    |   movel([0.113074, -1.368242, -2.579336, -0.764810, 1.570796, 1.683871],accel_mss,speed_ms,0,blend_radius_m)
    |   movel([0.112842, -1.368148, -2.579401, -0.764840, 1.570796, 1.683639],accel_mss,speed_ms,0,blend_radius_m)
    |   movel([0.112523, -1.368181, -2.579379, -0.764830, 1.570796, 1.683319],accel_mss,speed_ms,0,blend_radius_m)
    |   movel([0.111949, -1.368213, -2.579357, -0.764820, 1.570796, 1.682746],accel_mss,speed_ms,0,blend_radius_m)
    |   movel([0.111243, -1.367988, -2.579512, -0.764890, 1.570796, 1.682039],accel_mss,speed_ms,0,blend_radius_m)
    |   movel([0.110603, -1.367616, -2.579767, -0.765006, 1.570796, 1.681399],accel_mss,speed_ms,0,blend_radius_m)
    |   movel([0.110212, -1.367165, -2.580077, -0.765147, 1.570796, 1.681008],accel_mss,speed_ms,0,blend_radius_m)
    |   movel([0.110029, -1.366891, -2.580265, -0.765233, 1.570796, 1.680825],accel_mss,speed_ms,0,blend_radius_m)
    |   movel([0.109878, -1.366752, -2.580361, -0.765276, 1.570796, 1.680674],accel_mss,speed_ms,0,blend_radius_m)
    |   movel([0.109999, -1.366376, -2.580619, -0.765394, 1.570796, 1.680795],accel_mss,speed_ms,0,blend_radius_m)
    |   movel([0.110066, -1.366058, -2.580837, -0.765494, 1.570796, 1.680862],accel_mss,speed_ms,0,blend_radius_m)
    |   movel([0.110125, -1.365664, -2.581106, -0.765618, 1.570796, 1.680922],accel_mss,speed_ms,0,blend_radius_m)
    |   movel([0.110214, -1.365078, -2.581508, -0.765803, 1.570796, 1.681011],accel_mss,speed_ms,0,blend_radius_m)
    |   movel([0.110312, -1.364717, -2.581755, -0.765918, 1.570796, 1.681108],accel_mss,speed_ms,0,blend_radius_m)
    |   movel([0.110471, -1.364372, -2.581990, -0.766027, 1.570796, 1.681267],accel_mss,speed_ms,0,blend_radius_m)
    |   movel([0.110770, -1.363875, -2.582330, -0.766185, 1.570796, 1.681566],accel_mss,speed_ms,0,blend_radius_m)
    |   movel([0.111001, -1.363529, -2.582566, -0.766294, 1.570796, 1.681797],accel_mss,speed_ms,0,blend_radius_m)
    |   movel([0.111258, -1.363172, -2.582809, -0.766408, 1.570796, 1.682054],accel_mss,speed_ms,0,blend_radius_m)
    |   movel([0.111508, -1.362853, -2.583026, -0.766510, 1.570796, 1.682304],accel_mss,speed_ms,0,blend_radius_m)
    |   movel([0.111700, -1.362635, -2.583174, -0.766579, 1.570796, 1.682497],accel_mss,speed_ms,0,blend_radius_m)
    |   movel([0.112170, -1.362219, -2.583458, -0.766713, 1.570796, 1.682966],accel_mss,speed_ms,0,blend_radius_m)
    |   movel([0.112837, -1.361736, -2.583786, -0.766867, 1.570796, 1.683634],accel_mss,speed_ms,0,blend_radius_m)
    |   movel([0.113532, -1.361295, -2.584086, -0.767009, 1.570796, 1.684329],accel_mss,speed_ms,0,blend_radius_m)
    |   movel([0.114080, -1.361022, -2.584271, -0.767097, 1.570796, 1.684876],accel_mss,speed_ms,0,blend_radius_m)
    |   movel([0.114439, -1.360855, -2.584384, -0.767150, 1.570796, 1.685235],accel_mss,speed_ms,0,blend_radius_m)
    |   movel([0.114838, -1.360572, -2.584576, -0.767242, 1.570796, 1.685635],accel_mss,speed_ms,0,blend_radius_m)
    |   movel([0.115414, -1.360389, -2.584700, -0.767301, 1.570796, 1.686211],accel_mss,speed_ms,0,blend_radius_m)
    |   movel([0.115941, -1.360262, -2.584785, -0.767341, 1.570796, 1.686737],accel_mss,speed_ms,0,blend_radius_m)
    |   movel([0.116093, -1.360400, -2.584692, -0.767297, 1.570796, 1.686889],accel_mss,speed_ms,0,blend_radius_m)
    |   movel([0.116466, -1.360370, -2.584712, -0.767307, 1.570796, 1.687262],accel_mss,speed_ms,0,blend_radius_m)
    |   movel([0.117091, -1.360338, -2.584734, -0.767317, 1.570796, 1.687887],accel_mss,speed_ms,0,blend_radius_m)
    |   movel([0.117773, -1.360429, -2.584672, -0.767288, 1.570796, 1.688569],accel_mss,speed_ms,0,blend_radius_m)
    |   movel([0.118423, -1.360624, -2.584540, -0.767225, 1.570796, 1.689219],accel_mss,speed_ms,0,blend_radius_m)
    |   movel([0.118955, -1.360908, -2.584348, -0.767133, 1.570796, 1.689751],accel_mss,speed_ms,0,blend_radius_m)
    |   movel([0.119345, -1.361234, -2.584126, -0.767028, 1.570796, 1.690142],accel_mss,speed_ms,0,blend_radius_m)
    |   movel([0.119677, -1.361646, -2.583847, -0.766896, 1.570796, 1.690474],accel_mss,speed_ms,0,blend_radius_m)
    |   movel([0.119903, -1.362061, -2.583565, -0.766763, 1.570796, 1.690699],accel_mss,speed_ms,0,blend_radius_m)
    |   movel([0.119940, -1.362378, -2.583349, -0.766661, 1.570796, 1.690737],accel_mss,speed_ms,0,blend_radius_m)
    |   movel([0.119963, -1.362607, -2.583194, -0.766588, 1.570796, 1.690759],accel_mss,speed_ms,0,blend_radius_m)
    |   movel([0.120018, -1.362814, -2.583053, -0.766522, 1.570796, 1.690814],accel_mss,speed_ms,0,blend_radius_m)
    |   movel([0.119974, -1.363148, -2.582825, -0.766416, 1.570796, 1.690771],accel_mss,speed_ms,0,blend_radius_m)
    |   movel([0.119941, -1.363465, -2.582609, -0.766315, 1.570796, 1.690737],accel_mss,speed_ms,0,blend_radius_m)
    |   movel([0.120103, -1.363586, -2.582526, -0.766276, 1.570796, 1.690899],accel_mss,speed_ms,0,blend_radius_m)
    |   movel([0.120063, -1.363825, -2.582364, -0.766200, 1.570796, 1.690859],accel_mss,speed_ms,0,blend_radius_m)
    |   movel([0.119744, -1.364111, -2.582168, -0.766109, 1.570796, 1.690540],accel_mss,speed_ms,0,blend_radius_m)
    |   movel([0.119488, -1.364550, -2.581869, -0.765970, 1.570796, 1.690284],accel_mss,speed_ms,0,blend_radius_m)
    |   movel([0.118959, -1.365356, -2.581317, -0.765715, 1.570796, 1.689756],accel_mss,speed_ms,0,blend_radius_m)
    |   movel([0.118185, -1.366126, -2.580790, -0.765473, 1.570796, 1.688981],accel_mss,speed_ms,0,blend_radius_m)
    |   movel([0.117294, -1.366745, -2.580366, -0.765279, 1.570796, 1.688091],accel_mss,speed_ms,0,blend_radius_m)
    |   movel([0.116416, -1.367114, -2.580112, -0.765163, 1.570796, 1.687213],accel_mss,speed_ms,0,blend_radius_m)
    |   movel([0.116092, -1.367241, -2.580025, -0.765123, 1.570796, 1.686888],accel_mss,speed_ms,0,blend_radius_m)
    |   movel([0.115731, -1.367579, -2.579793, -0.765017, 1.570796, 1.686528],accel_mss,speed_ms,0,blend_radius_m)
    |   movel([0.115661, -1.367816, -2.579630, -0.764943, 1.570796, 1.686457],accel_mss,speed_ms,0,blend_radius_m)
    |   movel([0.115748, -1.368044, -2.579473, -0.764872, 1.570796, 1.686544],accel_mss,speed_ms,0,blend_radius_m)
    |   movel([0.115829, -1.368244, -2.579335, -0.764810, 1.570796, 1.686625],accel_mss,speed_ms,0,blend_radius_m)
    |   movel([0.115565, -1.368425, -2.579211, -0.764754, 1.570796, 1.686362],accel_mss,speed_ms,0,blend_radius_m)
    |   movel([0.115373, -1.368755, -2.578983, -0.764651, 1.570796, 1.686169],accel_mss,speed_ms,0,blend_radius_m)
    |   movel([0.115111, -1.368926, -2.578865, -0.764598, 1.570796, 1.685907],accel_mss,speed_ms,0,blend_radius_m)
    |   movel([0.114895, -1.368883, -2.578895, -0.764611, 1.570796, 1.685691],accel_mss,speed_ms,0,blend_radius_m)
    |   movel([0.114646, -1.368902, -2.578882, -0.764605, 1.570796, 1.685442],accel_mss,speed_ms,0,blend_radius_m)
    |   movel([0.114354, -1.368984, -2.578826, -0.764580, 1.570796, 1.685151],accel_mss,speed_ms,0,blend_radius_m)
    |   movel([0.114218, -1.368703, -2.579019, -0.764667, 1.570796, 1.685014],accel_mss,speed_ms,0,blend_radius_m)
    |   movel([0.114179, -1.368458, -2.579188, -0.764743, 1.570796, 1.684976],accel_mss,speed_ms,0,blend_radius_m)
    |   movel([0.113902, -1.368506, -2.579155, -0.764728, 1.570796, 1.684698],accel_mss,speed_ms,0,blend_radius_m)
    |   movel([0.113822, -1.368763, -2.578978, -0.764649, 1.570796, 1.684618],accel_mss,speed_ms,0,blend_radius_m)
    |   movel([0.113746, -1.369031, -2.578793, -0.764565, 1.570796, 1.684542],accel_mss,speed_ms,0,blend_radius_m)
    |   movel([0.113433, -1.369351, -2.578572, -0.764466, 1.570796, 1.684229],accel_mss,speed_ms,0,blend_radius_m)
    |   speed_ms = 0.003
    |   movel([0.113433, -1.372674, -2.580076, -0.759639, 1.570796, 1.684229],accel_mss,speed_ms,0,blend_radius_m)
    |   speed_ms = 0.007
    |   movel([0.113200, -1.372440, -2.580238, -0.759711, 1.570796, 1.683996],accel_mss,speed_ms,0,blend_radius_m)
    |   movel([0.113209, -1.372110, -2.580467, -0.759812, 1.570796, 1.684005],accel_mss,speed_ms,0,blend_radius_m)
    |   movel([0.113200, -1.371785, -2.580692, -0.759912, 1.570796, 1.683996],accel_mss,speed_ms,0,blend_radius_m)
    |   movel([0.113074, -1.371568, -2.580842, -0.759979, 1.570796, 1.683871],accel_mss,speed_ms,0,blend_radius_m)
    |   movel([0.112842, -1.371474, -2.580907, -0.760008, 1.570796, 1.683639],accel_mss,speed_ms,0,blend_radius_m)
    |   movel([0.112523, -1.371507, -2.580885, -0.759998, 1.570796, 1.683319],accel_mss,speed_ms,0,blend_radius_m)
    |   movel([0.111949, -1.371539, -2.580863, -0.759988, 1.570796, 1.682746],accel_mss,speed_ms,0,blend_radius_m)
    |   movel([0.111243, -1.371314, -2.581018, -0.760057, 1.570796, 1.682039],accel_mss,speed_ms,0,blend_radius_m)
    |   movel([0.110603, -1.370943, -2.581274, -0.760171, 1.570796, 1.681399],accel_mss,speed_ms,0,blend_radius_m)
    |   movel([0.110212, -1.370493, -2.581585, -0.760311, 1.570796, 1.681008],accel_mss,speed_ms,0,blend_radius_m)
    |   movel([0.110029, -1.370220, -2.581773, -0.760395, 1.570796, 1.680825],accel_mss,speed_ms,0,blend_radius_m)
    |   movel([0.109878, -1.370081, -2.581869, -0.760438, 1.570796, 1.680674],accel_mss,speed_ms,0,blend_radius_m)
    |   movel([0.109999, -1.369706, -2.582128, -0.760555, 1.570796, 1.680795],accel_mss,speed_ms,0,blend_radius_m)
    |   movel([0.110066, -1.369389, -2.582347, -0.760653, 1.570796, 1.680862],accel_mss,speed_ms,0,blend_radius_m)
    |   movel([0.110125, -1.368997, -2.582617, -0.760776, 1.570796, 1.680922],accel_mss,speed_ms,0,blend_radius_m)
    |   movel([0.110214, -1.368412, -2.583019, -0.760958, 1.570796, 1.681011],accel_mss,speed_ms,0,blend_radius_m)
    |   movel([0.110312, -1.368052, -2.583266, -0.761071, 1.570796, 1.681108],accel_mss,speed_ms,0,blend_radius_m)
    |   movel([0.110471, -1.367708, -2.583502, -0.761178, 1.570796, 1.681267],accel_mss,speed_ms,0,blend_radius_m)
    |   movel([0.110770, -1.367212, -2.583843, -0.761334, 1.570796, 1.681566],accel_mss,speed_ms,0,blend_radius_m)
    |   movel([0.111001, -1.366867, -2.584079, -0.761443, 1.570796, 1.681797],accel_mss,speed_ms,0,blend_radius_m)
    |   movel([0.111258, -1.366511, -2.584323, -0.761555, 1.570796, 1.682054],accel_mss,speed_ms,0,blend_radius_m)
    |   movel([0.111508, -1.366193, -2.584541, -0.761655, 1.570796, 1.682304],accel_mss,speed_ms,0,blend_radius_m)
    |   movel([0.111700, -1.365976, -2.584689, -0.761724, 1.570796, 1.682497],accel_mss,speed_ms,0,blend_radius_m)
    |   movel([0.112170, -1.365560, -2.584974, -0.761855, 1.570796, 1.682966],accel_mss,speed_ms,0,blend_radius_m)
    |   movel([0.112837, -1.365078, -2.585303, -0.762008, 1.570796, 1.683634],accel_mss,speed_ms,0,blend_radius_m)
    |   movel([0.113532, -1.364639, -2.585603, -0.762147, 1.570796, 1.684329],accel_mss,speed_ms,0,blend_radius_m)
    |   movel([0.114080, -1.364366, -2.585789, -0.762234, 1.570796, 1.684876],accel_mss,speed_ms,0,blend_radius_m)
    |   movel([0.114439, -1.364200, -2.585902, -0.762287, 1.570796, 1.685235],accel_mss,speed_ms,0,blend_radius_m)
    |   movel([0.114838, -1.363918, -2.586094, -0.762377, 1.570796, 1.685635],accel_mss,speed_ms,0,blend_radius_m)
    |   movel([0.115414, -1.363735, -2.586219, -0.762435, 1.570796, 1.686211],accel_mss,speed_ms,0,blend_radius_m)
    |   movel([0.115941, -1.363609, -2.586304, -0.762475, 1.570796, 1.686737],accel_mss,speed_ms,0,blend_radius_m)
    |   movel([0.116093, -1.363746, -2.586211, -0.762432, 1.570796, 1.686889],accel_mss,speed_ms,0,blend_radius_m)
    |   movel([0.116466, -1.363716, -2.586231, -0.762441, 1.570796, 1.687262],accel_mss,speed_ms,0,blend_radius_m)
    |   movel([0.117091, -1.363685, -2.586253, -0.762451, 1.570796, 1.687887],accel_mss,speed_ms,0,blend_radius_m)
    |   movel([0.117773, -1.363775, -2.586191, -0.762422, 1.570796, 1.688569],accel_mss,speed_ms,0,blend_radius_m)
    |   movel([0.118423, -1.363970, -2.586059, -0.762360, 1.570796, 1.689219],accel_mss,speed_ms,0,blend_radius_m)
    |   movel([0.118955, -1.364253, -2.585866, -0.762270, 1.570796, 1.689751],accel_mss,speed_ms,0,blend_radius_m)
    |   movel([0.119345, -1.364579, -2.585644, -0.762167, 1.570796, 1.690142],accel_mss,speed_ms,0,blend_radius_m)
    |   movel([0.119677, -1.364989, -2.585364, -0.762036, 1.570796, 1.690474],accel_mss,speed_ms,0,blend_radius_m)
    |   movel([0.119903, -1.365403, -2.585081, -0.761905, 1.570796, 1.690699],accel_mss,speed_ms,0,blend_radius_m)
    |   movel([0.119940, -1.365720, -2.584865, -0.761805, 1.570796, 1.690737],accel_mss,speed_ms,0,blend_radius_m)
    |   movel([0.119963, -1.365947, -2.584709, -0.761733, 1.570796, 1.690759],accel_mss,speed_ms,0,blend_radius_m)
    |   movel([0.120018, -1.366154, -2.584568, -0.761667, 1.570796, 1.690814],accel_mss,speed_ms,0,blend_radius_m)
    |   movel([0.119974, -1.366487, -2.584339, -0.761562, 1.570796, 1.690771],accel_mss,speed_ms,0,blend_radius_m)
    |   movel([0.119941, -1.366803, -2.584123, -0.761463, 1.570796, 1.690737],accel_mss,speed_ms,0,blend_radius_m)
    |   movel([0.120103, -1.366924, -2.584040, -0.761425, 1.570796, 1.690899],accel_mss,speed_ms,0,blend_radius_m)
    |   movel([0.120063, -1.367162, -2.583877, -0.761350, 1.570796, 1.690859],accel_mss,speed_ms,0,blend_radius_m)
    |   movel([0.119744, -1.367448, -2.583681, -0.761260, 1.570796, 1.690540],accel_mss,speed_ms,0,blend_radius_m)
    |   movel([0.119488, -1.367886, -2.583381, -0.761123, 1.570796, 1.690284],accel_mss,speed_ms,0,blend_radius_m)
    |   movel([0.118959, -1.368690, -2.582828, -0.760871, 1.570796, 1.689756],accel_mss,speed_ms,0,blend_radius_m)
    |   movel([0.118185, -1.369457, -2.582300, -0.760632, 1.570796, 1.688981],accel_mss,speed_ms,0,blend_radius_m)
    |   movel([0.117294, -1.370074, -2.581874, -0.760441, 1.570796, 1.688091],accel_mss,speed_ms,0,blend_radius_m)
    |   movel([0.116416, -1.370443, -2.581620, -0.760326, 1.570796, 1.687213],accel_mss,speed_ms,0,blend_radius_m)
    |   movel([0.116092, -1.370570, -2.581532, -0.760287, 1.570796, 1.686888],accel_mss,speed_ms,0,blend_radius_m)
    |   movel([0.115731, -1.370906, -2.581300, -0.760183, 1.570796, 1.686528],accel_mss,speed_ms,0,blend_radius_m)
    |   movel([0.115661, -1.371143, -2.581136, -0.760110, 1.570796, 1.686457],accel_mss,speed_ms,0,blend_radius_m)
    |   movel([0.115748, -1.371370, -2.580979, -0.760040, 1.570796, 1.686544],accel_mss,speed_ms,0,blend_radius_m)
    |   movel([0.115829, -1.371570, -2.580841, -0.759978, 1.570796, 1.686625],accel_mss,speed_ms,0,blend_radius_m)
    |   movel([0.115565, -1.371750, -2.580716, -0.759923, 1.570796, 1.686362],accel_mss,speed_ms,0,blend_radius_m)
    |   movel([0.115373, -1.372079, -2.580488, -0.759822, 1.570796, 1.686169],accel_mss,speed_ms,0,blend_radius_m)
    |   movel([0.115111, -1.372250, -2.580370, -0.759769, 1.570796, 1.685907],accel_mss,speed_ms,0,blend_radius_m)
    |   movel([0.114895, -1.372207, -2.580400, -0.759782, 1.570796, 1.685691],accel_mss,speed_ms,0,blend_radius_m)
    |   movel([0.114646, -1.372226, -2.580387, -0.759777, 1.570796, 1.685442],accel_mss,speed_ms,0,blend_radius_m)
    |   movel([0.114354, -1.372307, -2.580330, -0.759751, 1.570796, 1.685151],accel_mss,speed_ms,0,blend_radius_m)
    |   movel([0.114218, -1.372028, -2.580524, -0.759837, 1.570796, 1.685014],accel_mss,speed_ms,0,blend_radius_m)
    |   movel([0.114179, -1.371783, -2.580693, -0.759913, 1.570796, 1.684976],accel_mss,speed_ms,0,blend_radius_m)
    |   movel([0.113902, -1.371831, -2.580660, -0.759898, 1.570796, 1.684698],accel_mss,speed_ms,0,blend_radius_m)
    |   movel([0.113822, -1.372087, -2.580483, -0.759819, 1.570796, 1.684618],accel_mss,speed_ms,0,blend_radius_m)
    |   movel([0.113746, -1.372354, -2.580298, -0.759737, 1.570796, 1.684542],accel_mss,speed_ms,0,blend_radius_m)
    |   movel([0.113433, -1.372674, -2.580076, -0.759639, 1.570796, 1.684229],accel_mss,speed_ms,0,blend_radius_m)
    |   speed_ms = 0.003
    |   movel([0.113433, -1.359522, -2.574009, -0.778858, 1.570796, 1.684229],accel_mss,speed_ms,0,blend_radius_m)
    |   speed_ms = 1.000
    |   movel([0.113433, -1.334323, -2.561482, -0.816584, 1.570796, 1.684229],accel_mss,speed_ms,0,blend_radius_m)
    |   movel([0.114853, -1.333089, -2.562290, -0.817010, 1.570796, 1.685649],accel_mss,speed_ms,0,blend_radius_m)
    |   movel([0.114853, -1.358310, -2.574833, -0.779247, 1.570796, 1.685649],accel_mss,speed_ms,0,blend_radius_m)
    |   speed_ms = 0.003
    |   movel([0.114853, -1.368148, -2.579401, -0.764840, 1.570796, 1.685649],accel_mss,speed_ms,0,blend_radius_m)
    |   speed_ms = 0.007
    |   movel([0.114797, -1.367902, -2.579570, -0.764916, 1.570796, 1.685593],accel_mss,speed_ms,0,blend_radius_m)
    |   movel([0.114829, -1.367601, -2.579777, -0.765011, 1.570796, 1.685626],accel_mss,speed_ms,0,blend_radius_m)
    |   movel([0.114890, -1.367234, -2.580030, -0.765125, 1.570796, 1.685686],accel_mss,speed_ms,0,blend_radius_m)
    |   movel([0.115073, -1.366962, -2.580217, -0.765211, 1.570796, 1.685869],accel_mss,speed_ms,0,blend_radius_m)
    |   movel([0.115228, -1.367178, -2.580068, -0.765143, 1.570796, 1.686024],accel_mss,speed_ms,0,blend_radius_m)
    |   movel([0.115200, -1.367570, -2.579799, -0.765020, 1.570796, 1.685996],accel_mss,speed_ms,0,blend_radius_m)
    |   movel([0.115155, -1.367837, -2.579615, -0.764937, 1.570796, 1.685951],accel_mss,speed_ms,0,blend_radius_m)
    |   movel([0.115032, -1.368103, -2.579432, -0.764854, 1.570796, 1.685828],accel_mss,speed_ms,0,blend_radius_m)
    |   speed_ms = 0.003
    |   movel([0.114853, -1.371474, -2.580907, -0.760008, 1.570796, 1.685649],accel_mss,speed_ms,0,blend_radius_m)
    |   speed_ms = 0.007
    |   movel([0.114797, -1.371229, -2.581077, -0.760083, 1.570796, 1.685593],accel_mss,speed_ms,0,blend_radius_m)
    |   movel([0.114829, -1.370928, -2.581285, -0.760176, 1.570796, 1.685626],accel_mss,speed_ms,0,blend_radius_m)
    |   movel([0.114890, -1.370562, -2.581537, -0.760289, 1.570796, 1.685686],accel_mss,speed_ms,0,blend_radius_m)
    |   movel([0.115073, -1.370291, -2.581725, -0.760373, 1.570796, 1.685869],accel_mss,speed_ms,0,blend_radius_m)
    |   movel([0.115228, -1.370506, -2.581576, -0.760307, 1.570796, 1.686024],accel_mss,speed_ms,0,blend_radius_m)
    |   movel([0.115200, -1.370898, -2.581306, -0.760186, 1.570796, 1.685996],accel_mss,speed_ms,0,blend_radius_m)
    |   movel([0.115155, -1.371163, -2.581122, -0.760104, 1.570796, 1.685951],accel_mss,speed_ms,0,blend_radius_m)
    |   movel([0.115032, -1.371429, -2.580938, -0.760022, 1.570796, 1.685828],accel_mss,speed_ms,0,blend_radius_m)
    |   speed_ms = 0.003
    |   movel([0.114853, -1.358310, -2.574833, -0.779247, 1.570796, 1.685649],accel_mss,speed_ms,0,blend_radius_m)
    |   speed_ms = 1.000
    |   movel([0.114853, -1.333089, -2.562290, -0.817010, 1.570796, 1.685649],accel_mss,speed_ms,0,blend_radius_m)
    |   movel([0.115300, -1.331245, -2.563492, -0.817651, 1.570796, 1.686097],accel_mss,speed_ms,0,blend_radius_m)
    |   movel([0.115300, -1.356498, -2.576059, -0.779832, 1.570796, 1.686097],accel_mss,speed_ms,0,blend_radius_m)
    |   speed_ms = 0.003
    |   movel([0.115300, -1.366350, -2.580637, -0.765403, 1.570796, 1.686097],accel_mss,speed_ms,0,blend_radius_m)
    |   speed_ms = 0.007
    |   movel([0.115147, -1.366199, -2.580740, -0.765450, 1.570796, 1.685943],accel_mss,speed_ms,0,blend_radius_m)
    |   movel([0.115161, -1.365756, -2.581044, -0.765589, 1.570796, 1.685958],accel_mss,speed_ms,0,blend_radius_m)
    |   movel([0.114937, -1.365561, -2.581178, -0.765651, 1.570796, 1.685734],accel_mss,speed_ms,0,blend_radius_m)
    |   movel([0.114685, -1.365743, -2.581052, -0.765593, 1.570796, 1.685482],accel_mss,speed_ms,0,blend_radius_m)
    |   movel([0.114564, -1.365999, -2.580877, -0.765513, 1.570796, 1.685360],accel_mss,speed_ms,0,blend_radius_m)
    |   movel([0.114505, -1.366260, -2.580699, -0.765431, 1.570796, 1.685301],accel_mss,speed_ms,0,blend_radius_m)
    |   movel([0.114305, -1.366479, -2.580548, -0.765362, 1.570796, 1.685101],accel_mss,speed_ms,0,blend_radius_m)
    |   movel([0.114150, -1.366331, -2.580649, -0.765408, 1.570796, 1.684947],accel_mss,speed_ms,0,blend_radius_m)
    |   movel([0.114152, -1.365911, -2.580937, -0.765540, 1.570796, 1.684948],accel_mss,speed_ms,0,blend_radius_m)
    |   movel([0.114050, -1.365717, -2.581071, -0.765602, 1.570796, 1.684846],accel_mss,speed_ms,0,blend_radius_m)
    |   movel([0.113872, -1.365616, -2.581140, -0.765634, 1.570796, 1.684668],accel_mss,speed_ms,0,blend_radius_m)
    |   movel([0.113440, -1.365643, -2.581121, -0.765625, 1.570796, 1.684236],accel_mss,speed_ms,0,blend_radius_m)
    |   movel([0.113058, -1.365470, -2.581240, -0.765680, 1.570796, 1.683854],accel_mss,speed_ms,0,blend_radius_m)
    |   movel([0.112877, -1.365278, -2.581371, -0.765740, 1.570796, 1.683673],accel_mss,speed_ms,0,blend_radius_m)
    |   movel([0.112754, -1.365018, -2.581549, -0.765822, 1.570796, 1.683550],accel_mss,speed_ms,0,blend_radius_m)
    |   movel([0.112941, -1.364690, -2.581773, -0.765926, 1.570796, 1.683737],accel_mss,speed_ms,0,blend_radius_m)
    |   movel([0.113216, -1.364401, -2.581970, -0.766017, 1.570796, 1.684013],accel_mss,speed_ms,0,blend_radius_m)
    |   movel([0.113587, -1.364309, -2.582033, -0.766047, 1.570796, 1.684383],accel_mss,speed_ms,0,blend_radius_m)
    |   movel([0.113919, -1.364304, -2.582037, -0.766048, 1.570796, 1.684715],accel_mss,speed_ms,0,blend_radius_m)
    |   movel([0.114137, -1.364361, -2.581997, -0.766030, 1.570796, 1.684933],accel_mss,speed_ms,0,blend_radius_m)
    |   movel([0.114307, -1.364503, -2.581901, -0.765985, 1.570796, 1.685103],accel_mss,speed_ms,0,blend_radius_m)
    |   movel([0.114482, -1.364779, -2.581712, -0.765898, 1.570796, 1.685278],accel_mss,speed_ms,0,blend_radius_m)
    |   movel([0.114658, -1.365037, -2.581536, -0.765816, 1.570796, 1.685455],accel_mss,speed_ms,0,blend_radius_m)
    |   movel([0.114837, -1.365132, -2.581471, -0.765786, 1.570796, 1.685633],accel_mss,speed_ms,0,blend_radius_m)
    |   movel([0.115325, -1.364910, -2.581623, -0.765856, 1.570796, 1.686121],accel_mss,speed_ms,0,blend_radius_m)
    |   movel([0.115621, -1.364725, -2.581749, -0.765915, 1.570796, 1.686417],accel_mss,speed_ms,0,blend_radius_m)
    |   movel([0.115907, -1.364643, -2.581805, -0.765941, 1.570796, 1.686703],accel_mss,speed_ms,0,blend_radius_m)
    |   movel([0.116371, -1.364357, -2.582001, -0.766032, 1.570796, 1.687167],accel_mss,speed_ms,0,blend_radius_m)
    |   movel([0.116464, -1.364121, -2.582162, -0.766106, 1.570796, 1.687260],accel_mss,speed_ms,0,blend_radius_m)
    |   movel([0.116312, -1.363881, -2.582325, -0.766182, 1.570796, 1.687108],accel_mss,speed_ms,0,blend_radius_m)
    |   movel([0.116012, -1.364107, -2.582171, -0.766111, 1.570796, 1.686808],accel_mss,speed_ms,0,blend_radius_m)
    |   movel([0.115646, -1.364425, -2.581954, -0.766010, 1.570796, 1.686443],accel_mss,speed_ms,0,blend_radius_m)
    |   movel([0.115581, -1.364176, -2.582124, -0.766089, 1.570796, 1.686377],accel_mss,speed_ms,0,blend_radius_m)
    |   movel([0.115831, -1.363884, -2.582323, -0.766181, 1.570796, 1.686627],accel_mss,speed_ms,0,blend_radius_m)
    |   movel([0.116106, -1.363605, -2.582514, -0.766270, 1.570796, 1.686902],accel_mss,speed_ms,0,blend_radius_m)
    |   movel([0.116442, -1.363532, -2.582564, -0.766294, 1.570796, 1.687238],accel_mss,speed_ms,0,blend_radius_m)
    |   movel([0.116664, -1.363637, -2.582492, -0.766260, 1.570796, 1.687460],accel_mss,speed_ms,0,blend_radius_m)
    |   movel([0.116856, -1.363863, -2.582338, -0.766188, 1.570796, 1.687653],accel_mss,speed_ms,0,blend_radius_m)
    |   movel([0.116823, -1.364149, -2.582142, -0.766097, 1.570796, 1.687619],accel_mss,speed_ms,0,blend_radius_m)
    |   movel([0.116538, -1.364541, -2.581875, -0.765973, 1.570796, 1.687334],accel_mss,speed_ms,0,blend_radius_m)
    |   movel([0.115912, -1.365137, -2.581468, -0.765785, 1.570796, 1.686708],accel_mss,speed_ms,0,blend_radius_m)
    |   movel([0.115665, -1.365447, -2.581255, -0.765687, 1.570796, 1.686461],accel_mss,speed_ms,0,blend_radius_m)
    |   movel([0.115550, -1.365853, -2.580977, -0.765559, 1.570796, 1.686346],accel_mss,speed_ms,0,blend_radius_m)
    |   movel([0.115461, -1.366207, -2.580735, -0.765447, 1.570796, 1.686258],accel_mss,speed_ms,0,blend_radius_m)
    |   speed_ms = 0.003
    |   movel([0.115300, -1.369680, -2.582146, -0.760563, 1.570796, 1.686097],accel_mss,speed_ms,0,blend_radius_m)
    |   speed_ms = 0.007
    |   movel([0.115147, -1.369530, -2.582249, -0.760610, 1.570796, 1.685943],accel_mss,speed_ms,0,blend_radius_m)
    |   movel([0.115161, -1.369088, -2.582554, -0.760747, 1.570796, 1.685958],accel_mss,speed_ms,0,blend_radius_m)
    |   movel([0.114937, -1.368893, -2.582688, -0.760808, 1.570796, 1.685734],accel_mss,speed_ms,0,blend_radius_m)
    |   movel([0.114685, -1.369075, -2.582562, -0.760751, 1.570796, 1.685482],accel_mss,speed_ms,0,blend_radius_m)
    |   movel([0.114564, -1.369331, -2.582387, -0.760671, 1.570796, 1.685360],accel_mss,speed_ms,0,blend_radius_m)
    |   movel([0.114505, -1.369590, -2.582208, -0.760591, 1.570796, 1.685301],accel_mss,speed_ms,0,blend_radius_m)
    |   movel([0.114305, -1.369810, -2.582057, -0.760523, 1.570796, 1.685101],accel_mss,speed_ms,0,blend_radius_m)
    |   movel([0.114150, -1.369662, -2.582158, -0.760569, 1.570796, 1.684947],accel_mss,speed_ms,0,blend_radius_m)
    |   movel([0.114152, -1.369243, -2.582447, -0.760699, 1.570796, 1.684948],accel_mss,speed_ms,0,blend_radius_m)
    |   movel([0.114050, -1.369049, -2.582581, -0.760759, 1.570796, 1.684846],accel_mss,speed_ms,0,blend_radius_m)
    |   movel([0.113872, -1.368948, -2.582650, -0.760791, 1.570796, 1.684668],accel_mss,speed_ms,0,blend_radius_m)
    |   movel([0.113440, -1.368975, -2.582631, -0.760782, 1.570796, 1.684236],accel_mss,speed_ms,0,blend_radius_m)
    |   movel([0.113058, -1.368803, -2.582750, -0.760836, 1.570796, 1.683854],accel_mss,speed_ms,0,blend_radius_m)
    |   movel([0.112877, -1.368611, -2.582882, -0.760896, 1.570796, 1.683673],accel_mss,speed_ms,0,blend_radius_m)
    |   movel([0.112754, -1.368352, -2.583060, -0.760977, 1.570796, 1.683550],accel_mss,speed_ms,0,blend_radius_m)
    |   movel([0.112941, -1.368025, -2.583285, -0.761079, 1.570796, 1.683737],accel_mss,speed_ms,0,blend_radius_m)
    |   movel([0.113216, -1.367737, -2.583483, -0.761169, 1.570796, 1.684013],accel_mss,speed_ms,0,blend_radius_m)
    |   movel([0.113587, -1.367646, -2.583545, -0.761198, 1.570796, 1.684383],accel_mss,speed_ms,0,blend_radius_m)
    |   movel([0.113919, -1.367640, -2.583549, -0.761200, 1.570796, 1.684715],accel_mss,speed_ms,0,blend_radius_m)
    |   movel([0.114137, -1.367697, -2.583510, -0.761182, 1.570796, 1.684933],accel_mss,speed_ms,0,blend_radius_m)
    |   movel([0.114307, -1.367839, -2.583413, -0.761137, 1.570796, 1.685103],accel_mss,speed_ms,0,blend_radius_m)
    |   movel([0.114482, -1.368114, -2.583224, -0.761051, 1.570796, 1.685278],accel_mss,speed_ms,0,blend_radius_m)
    |   movel([0.114658, -1.368371, -2.583047, -0.760971, 1.570796, 1.685455],accel_mss,speed_ms,0,blend_radius_m)
    |   movel([0.114837, -1.368465, -2.582982, -0.760941, 1.570796, 1.685633],accel_mss,speed_ms,0,blend_radius_m)
    |   movel([0.115325, -1.368244, -2.583134, -0.761011, 1.570796, 1.686121],accel_mss,speed_ms,0,blend_radius_m)
    |   movel([0.115621, -1.368060, -2.583261, -0.761068, 1.570796, 1.686417],accel_mss,speed_ms,0,blend_radius_m)
    |   movel([0.115907, -1.367978, -2.583317, -0.761094, 1.570796, 1.686703],accel_mss,speed_ms,0,blend_radius_m)
    |   movel([0.116371, -1.367693, -2.583513, -0.761183, 1.570796, 1.687167],accel_mss,speed_ms,0,blend_radius_m)
    |   movel([0.116464, -1.367457, -2.583675, -0.761257, 1.570796, 1.687260],accel_mss,speed_ms,0,blend_radius_m)
    |   movel([0.116312, -1.367218, -2.583838, -0.761332, 1.570796, 1.687108],accel_mss,speed_ms,0,blend_radius_m)
    |   movel([0.116012, -1.367444, -2.583684, -0.761261, 1.570796, 1.686808],accel_mss,speed_ms,0,blend_radius_m)
    |   movel([0.115646, -1.367760, -2.583467, -0.761162, 1.570796, 1.686443],accel_mss,speed_ms,0,blend_radius_m)
    |   movel([0.115581, -1.367513, -2.583637, -0.761240, 1.570796, 1.686377],accel_mss,speed_ms,0,blend_radius_m)
    |   movel([0.115831, -1.367222, -2.583836, -0.761331, 1.570796, 1.686627],accel_mss,speed_ms,0,blend_radius_m)
    |   movel([0.116106, -1.366943, -2.584028, -0.761419, 1.570796, 1.686902],accel_mss,speed_ms,0,blend_radius_m)
    |   movel([0.116442, -1.366870, -2.584077, -0.761442, 1.570796, 1.687238],accel_mss,speed_ms,0,blend_radius_m)
    |   movel([0.116664, -1.366974, -2.584006, -0.761409, 1.570796, 1.687460],accel_mss,speed_ms,0,blend_radius_m)
    |   movel([0.116856, -1.367200, -2.583851, -0.761338, 1.570796, 1.687653],accel_mss,speed_ms,0,blend_radius_m)
    |   movel([0.116823, -1.367486, -2.583655, -0.761248, 1.570796, 1.687619],accel_mss,speed_ms,0,blend_radius_m)
    |   movel([0.116538, -1.367876, -2.583387, -0.761126, 1.570796, 1.687334],accel_mss,speed_ms,0,blend_radius_m)
    |   movel([0.115912, -1.368471, -2.582979, -0.760940, 1.570796, 1.686708],accel_mss,speed_ms,0,blend_radius_m)
    |   movel([0.115665, -1.368780, -2.582766, -0.760843, 1.570796, 1.686461],accel_mss,speed_ms,0,blend_radius_m)
    |   movel([0.115550, -1.369185, -2.582487, -0.760717, 1.570796, 1.686346],accel_mss,speed_ms,0,blend_radius_m)
    |   movel([0.115461, -1.369538, -2.582244, -0.760607, 1.570796, 1.686258],accel_mss,speed_ms,0,blend_radius_m)
    |   speed_ms = 0.003
    |   movel([0.115300, -1.356498, -2.576059, -0.779832, 1.570796, 1.686097],accel_mss,speed_ms,0,blend_radius_m)
    |   speed_ms = 1.000
    |   movel([0.115300, -1.331245, -2.563492, -0.817651, 1.570796, 1.686097],accel_mss,speed_ms,0,blend_radius_m)
    |   movel([0.114036, -1.330032, -2.564282, -0.818075, 1.570796, 1.684833],accel_mss,speed_ms,0,blend_radius_m)
    |   movel([0.114036, -1.355305, -2.576864, -0.780220, 1.570796, 1.684833],accel_mss,speed_ms,0,blend_radius_m)
    |   speed_ms = 0.003
    |   movel([0.114036, -1.365165, -2.581448, -0.765776, 1.570796, 1.684833],accel_mss,speed_ms,0,blend_radius_m)
    |   speed_ms = 0.007
    |   movel([0.113723, -1.365329, -2.581336, -0.765724, 1.570796, 1.684520],accel_mss,speed_ms,0,blend_radius_m)
    |   movel([0.113357, -1.365280, -2.581370, -0.765739, 1.570796, 1.684153],accel_mss,speed_ms,0,blend_radius_m)
    |   movel([0.113127, -1.365067, -2.581515, -0.765807, 1.570796, 1.683924],accel_mss,speed_ms,0,blend_radius_m)
    |   movel([0.113178, -1.364791, -2.581704, -0.765894, 1.570796, 1.683974],accel_mss,speed_ms,0,blend_radius_m)
    |   movel([0.113608, -1.364574, -2.581852, -0.765963, 1.570796, 1.684405],accel_mss,speed_ms,0,blend_radius_m)
    |   movel([0.113870, -1.364583, -2.581846, -0.765960, 1.570796, 1.684666],accel_mss,speed_ms,0,blend_radius_m)
    |   movel([0.114043, -1.364683, -2.581778, -0.765928, 1.570796, 1.684839],accel_mss,speed_ms,0,blend_radius_m)
    |   movel([0.114163, -1.364837, -2.581673, -0.765879, 1.570796, 1.684959],accel_mss,speed_ms,0,blend_radius_m)
    |   movel([0.114036, -1.365165, -2.581448, -0.765776, 1.570796, 1.684833],accel_mss,speed_ms,0,blend_radius_m)
    |   speed_ms = 0.003
    |   movel([0.114036, -1.368499, -2.582959, -0.760931, 1.570796, 1.684833],accel_mss,speed_ms,0,blend_radius_m)
    |   speed_ms = 0.007
    |   movel([0.113723, -1.368662, -2.582847, -0.760880, 1.570796, 1.684520],accel_mss,speed_ms,0,blend_radius_m)
    |   movel([0.113357, -1.368613, -2.582880, -0.760895, 1.570796, 1.684153],accel_mss,speed_ms,0,blend_radius_m)
    |   movel([0.113127, -1.368401, -2.583026, -0.760962, 1.570796, 1.683924],accel_mss,speed_ms,0,blend_radius_m)
    |   movel([0.113178, -1.368126, -2.583215, -0.761047, 1.570796, 1.683974],accel_mss,speed_ms,0,blend_radius_m)
    |   movel([0.113608, -1.367909, -2.583364, -0.761115, 1.570796, 1.684405],accel_mss,speed_ms,0,blend_radius_m)
    |   movel([0.113870, -1.367919, -2.583358, -0.761112, 1.570796, 1.684666],accel_mss,speed_ms,0,blend_radius_m)
    |   movel([0.114043, -1.368018, -2.583289, -0.761081, 1.570796, 1.684839],accel_mss,speed_ms,0,blend_radius_m)
    |   movel([0.114163, -1.368172, -2.583184, -0.761033, 1.570796, 1.684959],accel_mss,speed_ms,0,blend_radius_m)
    |   movel([0.114036, -1.368499, -2.582959, -0.760931, 1.570796, 1.684833],accel_mss,speed_ms,0,blend_radius_m)
    |   speed_ms = 0.003
    |   movel([0.114036, -1.355305, -2.576864, -0.780220, 1.570796, 1.684833],accel_mss,speed_ms,0,blend_radius_m)
    |   speed_ms = 1.000
    |   movel([0.114036, -1.330032, -2.564282, -0.818075, 1.570796, 1.684833],accel_mss,speed_ms,0,blend_radius_m)
    |   movel([0.107334, -1.332493, -2.562679, -0.817217, 1.570796, 1.678130],accel_mss,speed_ms,0,blend_radius_m)
    |   movel([0.107334, -1.357724, -2.575230, -0.779436, 1.570796, 1.678130],accel_mss,speed_ms,0,blend_radius_m)
    |   speed_ms = 0.003
    |   movel([0.107334, -1.367566, -2.579801, -0.765021, 1.570796, 1.678130],accel_mss,speed_ms,0,blend_radius_m)
    |   speed_ms = 0.007
    |   movel([0.107250, -1.368281, -2.579310, -0.764798, 1.570796, 1.678047],accel_mss,speed_ms,0,blend_radius_m)
    |   movel([0.107024, -1.368666, -2.579044, -0.764679, 1.570796, 1.677820],accel_mss,speed_ms,0,blend_radius_m)
    |   movel([0.106591, -1.369021, -2.578799, -0.764568, 1.570796, 1.677388],accel_mss,speed_ms,0,blend_radius_m)
    |   movel([0.105893, -1.369496, -2.578472, -0.764421, 1.570796, 1.676689],accel_mss,speed_ms,0,blend_radius_m)
    |   movel([0.105181, -1.369942, -2.578164, -0.764283, 1.570796, 1.675977],accel_mss,speed_ms,0,blend_radius_m)
    |   movel([0.104870, -1.369983, -2.578136, -0.764270, 1.570796, 1.675666],accel_mss,speed_ms,0,blend_radius_m)
    |   movel([0.104761, -1.369797, -2.578264, -0.764328, 1.570796, 1.675557],accel_mss,speed_ms,0,blend_radius_m)
    |   movel([0.104653, -1.368422, -2.579213, -0.764755, 1.570796, 1.675449],accel_mss,speed_ms,0,blend_radius_m)
    |   movel([0.104510, -1.367756, -2.579671, -0.764962, 1.570796, 1.675306],accel_mss,speed_ms,0,blend_radius_m)
    |   movel([0.104276, -1.367419, -2.579903, -0.765067, 1.570796, 1.675072],accel_mss,speed_ms,0,blend_radius_m)
    |   movel([0.103915, -1.367320, -2.579970, -0.765098, 1.570796, 1.674711],accel_mss,speed_ms,0,blend_radius_m)
    |   movel([0.103332, -1.367539, -2.579820, -0.765030, 1.570796, 1.674129],accel_mss,speed_ms,0,blend_radius_m)
    |   movel([0.102835, -1.367799, -2.579641, -0.764949, 1.570796, 1.673632],accel_mss,speed_ms,0,blend_radius_m)
    |   movel([0.102185, -1.368173, -2.579384, -0.764832, 1.570796, 1.672982],accel_mss,speed_ms,0,blend_radius_m)
    |   movel([0.099075, -1.369824, -2.578246, -0.764320, 1.570796, 1.669871],accel_mss,speed_ms,0,blend_radius_m)
    |   movel([0.095590, -1.371345, -2.577193, -0.763851, 1.570796, 1.666387],accel_mss,speed_ms,0,blend_radius_m)
    |   movel([0.091812, -1.372711, -2.576245, -0.763432, 1.570796, 1.662609],accel_mss,speed_ms,0,blend_radius_m)
    |   movel([0.087807, -1.373897, -2.575421, -0.763072, 1.570796, 1.658604],accel_mss,speed_ms,0,blend_radius_m)
    |   movel([0.084957, -1.374600, -2.574930, -0.762858, 1.570796, 1.655753],accel_mss,speed_ms,0,blend_radius_m)
    |   movel([0.082581, -1.375066, -2.574606, -0.762718, 1.570796, 1.653377],accel_mss,speed_ms,0,blend_radius_m)
    |   movel([0.080422, -1.375336, -2.574417, -0.762636, 1.570796, 1.651219],accel_mss,speed_ms,0,blend_radius_m)
    |   movel([0.078241, -1.375448, -2.574339, -0.762603, 1.570796, 1.649037],accel_mss,speed_ms,0,blend_radius_m)
    |   movel([0.077595, -1.375463, -2.574328, -0.762598, 1.570796, 1.648391],accel_mss,speed_ms,0,blend_radius_m)
    |   movel([0.077017, -1.375486, -2.574312, -0.762591, 1.570796, 1.647813],accel_mss,speed_ms,0,blend_radius_m)
    |   movel([0.076527, -1.375514, -2.574293, -0.762583, 1.570796, 1.647323],accel_mss,speed_ms,0,blend_radius_m)
    |   movel([0.076144, -1.375675, -2.574180, -0.762534, 1.570796, 1.646941],accel_mss,speed_ms,0,blend_radius_m)
    |   movel([0.075861, -1.375963, -2.573979, -0.762448, 1.570796, 1.646658],accel_mss,speed_ms,0,blend_radius_m)
    |   movel([0.075599, -1.376321, -2.573728, -0.762340, 1.570796, 1.646396],accel_mss,speed_ms,0,blend_radius_m)
    |   movel([0.075421, -1.376678, -2.573478, -0.762233, 1.570796, 1.646217],accel_mss,speed_ms,0,blend_radius_m)
    |   movel([0.075249, -1.377242, -2.573082, -0.762064, 1.570796, 1.646045],accel_mss,speed_ms,0,blend_radius_m)
    |   movel([0.075143, -1.377642, -2.572802, -0.761945, 1.570796, 1.645939],accel_mss,speed_ms,0,blend_radius_m)
    |   movel([0.075046, -1.378040, -2.572523, -0.761826, 1.570796, 1.645843],accel_mss,speed_ms,0,blend_radius_m)
    |   movel([0.074952, -1.378421, -2.572255, -0.761713, 1.570796, 1.645748],accel_mss,speed_ms,0,blend_radius_m)
    |   movel([0.074853, -1.378765, -2.572013, -0.761611, 1.570796, 1.645650],accel_mss,speed_ms,0,blend_radius_m)
    |   movel([0.074757, -1.379053, -2.571810, -0.761526, 1.570796, 1.645554],accel_mss,speed_ms,0,blend_radius_m)
    |   movel([0.074468, -1.379289, -2.571644, -0.761456, 1.570796, 1.645264],accel_mss,speed_ms,0,blend_radius_m)
    |   movel([0.073765, -1.379305, -2.571633, -0.761451, 1.570796, 1.644562],accel_mss,speed_ms,0,blend_radius_m)
    |   movel([0.073075, -1.379262, -2.571663, -0.761464, 1.570796, 1.643871],accel_mss,speed_ms,0,blend_radius_m)
    |   movel([0.072682, -1.379139, -2.571750, -0.761500, 1.570796, 1.643478],accel_mss,speed_ms,0,blend_radius_m)
    |   movel([0.072546, -1.379010, -2.571840, -0.761538, 1.570796, 1.643342],accel_mss,speed_ms,0,blend_radius_m)
    |   movel([0.072521, -1.378523, -2.572183, -0.761683, 1.570796, 1.643318],accel_mss,speed_ms,0,blend_radius_m)
    |   movel([0.072656, -1.377720, -2.572748, -0.761922, 1.570796, 1.643452],accel_mss,speed_ms,0,blend_radius_m)
    |   movel([0.073767, -1.373164, -2.575931, -0.763294, 1.570796, 1.644564],accel_mss,speed_ms,0,blend_radius_m)
    |   movel([0.075488, -1.368756, -2.578983, -0.764651, 1.570796, 1.646285],accel_mss,speed_ms,0,blend_radius_m)
    |   movel([0.077718, -1.364727, -2.581747, -0.765914, 1.570796, 1.648514],accel_mss,speed_ms,0,blend_radius_m)
    |   movel([0.080351, -1.361316, -2.584071, -0.767002, 1.570796, 1.651147],accel_mss,speed_ms,0,blend_radius_m)
    |   movel([0.082795, -1.358951, -2.585672, -0.767766, 1.570796, 1.653591],accel_mss,speed_ms,0,blend_radius_m)
    |   movel([0.085385, -1.357041, -2.586960, -0.768389, 1.570796, 1.656181],accel_mss,speed_ms,0,blend_radius_m)
    |   movel([0.088218, -1.355526, -2.587977, -0.768886, 1.570796, 1.659014],accel_mss,speed_ms,0,blend_radius_m)
    |   movel([0.091400, -1.354347, -2.588767, -0.769275, 1.570796, 1.662196],accel_mss,speed_ms,0,blend_radius_m)
    |   movel([0.094574, -1.353626, -2.589249, -0.769514, 1.570796, 1.665370],accel_mss,speed_ms,0,blend_radius_m)
    |   movel([0.097379, -1.353476, -2.589349, -0.769564, 1.570796, 1.668175],accel_mss,speed_ms,0,blend_radius_m)
    |   movel([0.099838, -1.353910, -2.589059, -0.769420, 1.570796, 1.670634],accel_mss,speed_ms,0,blend_radius_m)
    |   movel([0.101993, -1.354916, -2.588386, -0.769087, 1.570796, 1.672790],accel_mss,speed_ms,0,blend_radius_m)
    |   movel([0.103899, -1.356588, -2.587264, -0.768537, 1.570796, 1.674695],accel_mss,speed_ms,0,blend_radius_m)
    |   movel([0.105421, -1.358873, -2.585725, -0.767791, 1.570796, 1.676217],accel_mss,speed_ms,0,blend_radius_m)
    |   movel([0.106518, -1.361692, -2.583816, -0.766881, 1.570796, 1.677314],accel_mss,speed_ms,0,blend_radius_m)
    |   movel([0.107156, -1.364956, -2.581591, -0.765842, 1.570796, 1.677952],accel_mss,speed_ms,0,blend_radius_m)
    |   movel([0.107310, -1.366526, -2.580516, -0.765347, 1.570796, 1.678107],accel_mss,speed_ms,0,blend_radius_m)
    |   movel([0.107334, -1.367566, -2.579801, -0.765021, 1.570796, 1.678130],accel_mss,speed_ms,0,blend_radius_m)
    |   speed_ms = 0.003
    |   movel([0.107334, -1.370894, -2.581308, -0.760187, 1.570796, 1.678130],accel_mss,speed_ms,0,blend_radius_m)
    |   speed_ms = 0.007
    |   movel([0.107250, -1.371606, -2.580816, -0.759967, 1.570796, 1.678047],accel_mss,speed_ms,0,blend_radius_m)
    |   movel([0.107024, -1.371990, -2.580550, -0.759849, 1.570796, 1.677820],accel_mss,speed_ms,0,blend_radius_m)
    |   movel([0.106591, -1.372345, -2.580304, -0.759740, 1.570796, 1.677388],accel_mss,speed_ms,0,blend_radius_m)
    |   movel([0.105893, -1.372818, -2.579976, -0.759595, 1.570796, 1.676689],accel_mss,speed_ms,0,blend_radius_m)
    |   movel([0.105181, -1.373264, -2.579667, -0.759459, 1.570796, 1.675977],accel_mss,speed_ms,0,blend_radius_m)
    |   movel([0.104870, -1.373304, -2.579639, -0.759446, 1.570796, 1.675666],accel_mss,speed_ms,0,blend_radius_m)
    |   movel([0.104761, -1.373118, -2.579768, -0.759503, 1.570796, 1.675557],accel_mss,speed_ms,0,blend_radius_m)
    |   movel([0.104653, -1.371747, -2.580718, -0.759924, 1.570796, 1.675449],accel_mss,speed_ms,0,blend_radius_m)
    |   movel([0.104510, -1.371083, -2.581178, -0.760128, 1.570796, 1.675306],accel_mss,speed_ms,0,blend_radius_m)
    |   movel([0.104276, -1.370747, -2.581410, -0.760232, 1.570796, 1.675072],accel_mss,speed_ms,0,blend_radius_m)
    |   movel([0.103915, -1.370648, -2.581478, -0.760263, 1.570796, 1.674711],accel_mss,speed_ms,0,blend_radius_m)
    |   movel([0.103332, -1.370866, -2.581327, -0.760195, 1.570796, 1.674129],accel_mss,speed_ms,0,blend_radius_m)
    |   movel([0.102835, -1.371126, -2.581148, -0.760115, 1.570796, 1.673632],accel_mss,speed_ms,0,blend_radius_m)
    |   movel([0.102185, -1.371499, -2.580890, -0.760000, 1.570796, 1.672982],accel_mss,speed_ms,0,blend_radius_m)
    |   movel([0.099075, -1.373145, -2.579749, -0.759495, 1.570796, 1.669871],accel_mss,speed_ms,0,blend_radius_m)
    |   movel([0.095590, -1.374663, -2.578694, -0.759032, 1.570796, 1.666387],accel_mss,speed_ms,0,blend_radius_m)
    |   movel([0.091812, -1.376025, -2.577744, -0.758620, 1.570796, 1.662609],accel_mss,speed_ms,0,blend_radius_m)
    |   movel([0.087807, -1.377207, -2.576917, -0.758264, 1.570796, 1.658604],accel_mss,speed_ms,0,blend_radius_m)
    |   movel([0.084957, -1.377909, -2.576426, -0.758054, 1.570796, 1.655753],accel_mss,speed_ms,0,blend_radius_m)
    |   movel([0.082581, -1.378373, -2.576100, -0.757916, 1.570796, 1.653377],accel_mss,speed_ms,0,blend_radius_m)
    |   movel([0.080422, -1.378642, -2.575911, -0.757835, 1.570796, 1.651219],accel_mss,speed_ms,0,blend_radius_m)
    |   movel([0.078241, -1.378754, -2.575833, -0.757802, 1.570796, 1.649037],accel_mss,speed_ms,0,blend_radius_m)
    |   movel([0.077595, -1.378769, -2.575822, -0.757798, 1.570796, 1.648391],accel_mss,speed_ms,0,blend_radius_m)
    |   movel([0.077017, -1.378792, -2.575806, -0.757791, 1.570796, 1.647813],accel_mss,speed_ms,0,blend_radius_m)
    |   movel([0.076527, -1.378820, -2.575787, -0.757783, 1.570796, 1.647323],accel_mss,speed_ms,0,blend_radius_m)
    |   movel([0.076144, -1.378981, -2.575673, -0.757735, 1.570796, 1.646941],accel_mss,speed_ms,0,blend_radius_m)
    |   movel([0.075861, -1.379268, -2.575472, -0.757649, 1.570796, 1.646658],accel_mss,speed_ms,0,blend_radius_m)
    |   movel([0.075599, -1.379625, -2.575220, -0.757543, 1.570796, 1.646396],accel_mss,speed_ms,0,blend_radius_m)
    |   movel([0.075421, -1.379981, -2.574970, -0.757438, 1.570796, 1.646217],accel_mss,speed_ms,0,blend_radius_m)
    |   movel([0.075249, -1.380544, -2.574573, -0.757272, 1.570796, 1.646045],accel_mss,speed_ms,0,blend_radius_m)
    |   movel([0.075143, -1.380942, -2.574293, -0.757154, 1.570796, 1.645939],accel_mss,speed_ms,0,blend_radius_m)
    |   movel([0.075046, -1.381339, -2.574012, -0.757037, 1.570796, 1.645843],accel_mss,speed_ms,0,blend_radius_m)
    |   movel([0.074952, -1.381719, -2.573744, -0.756926, 1.570796, 1.645748],accel_mss,speed_ms,0,blend_radius_m)
    |   movel([0.074853, -1.382062, -2.573502, -0.756825, 1.570796, 1.645650],accel_mss,speed_ms,0,blend_radius_m)
    |   movel([0.074757, -1.382350, -2.573298, -0.756741, 1.570796, 1.645554],accel_mss,speed_ms,0,blend_radius_m)
    |   movel([0.074468, -1.382585, -2.573132, -0.756672, 1.570796, 1.645264],accel_mss,speed_ms,0,blend_radius_m)
    |   movel([0.073765, -1.382601, -2.573121, -0.756668, 1.570796, 1.644562],accel_mss,speed_ms,0,blend_radius_m)
    |   movel([0.073075, -1.382558, -2.573151, -0.756680, 1.570796, 1.643871],accel_mss,speed_ms,0,blend_radius_m)
    |   movel([0.072682, -1.382435, -2.573238, -0.756716, 1.570796, 1.643478],accel_mss,speed_ms,0,blend_radius_m)
    |   movel([0.072546, -1.382307, -2.573329, -0.756753, 1.570796, 1.643342],accel_mss,speed_ms,0,blend_radius_m)
    |   movel([0.072521, -1.381821, -2.573672, -0.756896, 1.570796, 1.643318],accel_mss,speed_ms,0,blend_radius_m)
    |   movel([0.072656, -1.381020, -2.574238, -0.757131, 1.570796, 1.643452],accel_mss,speed_ms,0,blend_radius_m)
    |   movel([0.073767, -1.376476, -2.577429, -0.758484, 1.570796, 1.644564],accel_mss,speed_ms,0,blend_radius_m)
    |   movel([0.075488, -1.372080, -2.580488, -0.759821, 1.570796, 1.646285],accel_mss,speed_ms,0,blend_radius_m)
    |   movel([0.077718, -1.368062, -2.583259, -0.761067, 1.570796, 1.648514],accel_mss,speed_ms,0,blend_radius_m)
    |   movel([0.080351, -1.364660, -2.585588, -0.762141, 1.570796, 1.651147],accel_mss,speed_ms,0,blend_radius_m)
    |   movel([0.082795, -1.362302, -2.587193, -0.762894, 1.570796, 1.653591],accel_mss,speed_ms,0,blend_radius_m)
    |   movel([0.085385, -1.360396, -2.588484, -0.763509, 1.570796, 1.656181],accel_mss,speed_ms,0,blend_radius_m)
    |   movel([0.088218, -1.358885, -2.589504, -0.764000, 1.570796, 1.659014],accel_mss,speed_ms,0,blend_radius_m)
    |   movel([0.091400, -1.357709, -2.590296, -0.764384, 1.570796, 1.662196],accel_mss,speed_ms,0,blend_radius_m)
    |   movel([0.094574, -1.356990, -2.590779, -0.764620, 1.570796, 1.665370],accel_mss,speed_ms,0,blend_radius_m)
    |   movel([0.097379, -1.356841, -2.590879, -0.764669, 1.570796, 1.668175],accel_mss,speed_ms,0,blend_radius_m)
    |   movel([0.099838, -1.357273, -2.590589, -0.764527, 1.570796, 1.670634],accel_mss,speed_ms,0,blend_radius_m)
    |   movel([0.101993, -1.358277, -2.589914, -0.764198, 1.570796, 1.672790],accel_mss,speed_ms,0,blend_radius_m)
    |   movel([0.103899, -1.359945, -2.588789, -0.763655, 1.570796, 1.674695],accel_mss,speed_ms,0,blend_radius_m)
    |   movel([0.105421, -1.362224, -2.587246, -0.762919, 1.570796, 1.676217],accel_mss,speed_ms,0,blend_radius_m)
    |   movel([0.106518, -1.365035, -2.585333, -0.762022, 1.570796, 1.677314],accel_mss,speed_ms,0,blend_radius_m)
    |   movel([0.107156, -1.368290, -2.583103, -0.760996, 1.570796, 1.677952],accel_mss,speed_ms,0,blend_radius_m)
    |   movel([0.107310, -1.369856, -2.582025, -0.760508, 1.570796, 1.678107],accel_mss,speed_ms,0,blend_radius_m)
    |   movel([0.107334, -1.370894, -2.581308, -0.760187, 1.570796, 1.678130],accel_mss,speed_ms,0,blend_radius_m)
    |   speed_ms = 0.003
    |   movel([0.107334, -1.357724, -2.575230, -0.779436, 1.570796, 1.678130],accel_mss,speed_ms,0,blend_radius_m)
    |   speed_ms = 1.000
    |   movel([0.107334, -1.332493, -2.562679, -0.817217, 1.570796, 1.678130],accel_mss,speed_ms,0,blend_radius_m)
    |   movel([0.108777, -1.323962, -2.568202, -0.820226, 1.570796, 1.679573],accel_mss,speed_ms,0,blend_radius_m)
    |   movel([0.108777, -1.349338, -2.580862, -0.782189, 1.570796, 1.679573],accel_mss,speed_ms,0,blend_radius_m)
    |   speed_ms = 0.003
    |   movel([0.108777, -1.359243, -2.585475, -0.767671, 1.570796, 1.679573],accel_mss,speed_ms,0,blend_radius_m)
    |   speed_ms = 0.007
    |   speed_ms = 0.003
    |   movel([0.108777, -1.362592, -2.586996, -0.762801, 1.570796, 1.679573],accel_mss,speed_ms,0,blend_radius_m)
    |   speed_ms = 0.007
    |   speed_ms = 0.003
    |   movel([0.108777, -1.349338, -2.580862, -0.782189, 1.570796, 1.679573],accel_mss,speed_ms,0,blend_radius_m)
    |   speed_ms = 1.000
    |   movel([0.108777, -1.323962, -2.568202, -0.820226, 1.570796, 1.679573],accel_mss,speed_ms,0,blend_radius_m)
    |   movel([0.115883, -1.313834, -2.574634, -0.823920, 1.570796, 1.686679],accel_mss,speed_ms,0,blend_radius_m)
    |   movel([0.115883, -1.339378, -2.587426, -0.785585, 1.570796, 1.686679],accel_mss,speed_ms,0,blend_radius_m)
    |   speed_ms = 0.003
    |   movel([0.115883, -1.349357, -2.592088, -0.770944, 1.570796, 1.686679],accel_mss,speed_ms,0,blend_radius_m)
    |   speed_ms = 0.007
    |   movel([0.115699, -1.349014, -2.592315, -0.771060, 1.570796, 1.686495],accel_mss,speed_ms,0,blend_radius_m)
    |   movel([0.115676, -1.348698, -2.592524, -0.771167, 1.570796, 1.686472],accel_mss,speed_ms,0,blend_radius_m)
    |   movel([0.115575, -1.348533, -2.592633, -0.771223, 1.570796, 1.686372],accel_mss,speed_ms,0,blend_radius_m)
    |   movel([0.115017, -1.348527, -2.592637, -0.771225, 1.570796, 1.685813],accel_mss,speed_ms,0,blend_radius_m)
    |   movel([0.114668, -1.348560, -2.592615, -0.771214, 1.570796, 1.685464],accel_mss,speed_ms,0,blend_radius_m)
    |   movel([0.114704, -1.348286, -2.592796, -0.771307, 1.570796, 1.685500],accel_mss,speed_ms,0,blend_radius_m)
    |   movel([0.115071, -1.348116, -2.592908, -0.771365, 1.570796, 1.685867],accel_mss,speed_ms,0,blend_radius_m)
    |   movel([0.115442, -1.347956, -2.593014, -0.771419, 1.570796, 1.686238],accel_mss,speed_ms,0,blend_radius_m)
    |   movel([0.115828, -1.347543, -2.593286, -0.771560, 1.570796, 1.686625],accel_mss,speed_ms,0,blend_radius_m)
    |   movel([0.115940, -1.347188, -2.593520, -0.771680, 1.570796, 1.686737],accel_mss,speed_ms,0,blend_radius_m)
    |   movel([0.116063, -1.346865, -2.593733, -0.771791, 1.570796, 1.686859],accel_mss,speed_ms,0,blend_radius_m)
    |   movel([0.116375, -1.346777, -2.593791, -0.771821, 1.570796, 1.687171],accel_mss,speed_ms,0,blend_radius_m)
    |   movel([0.116418, -1.347053, -2.593609, -0.771727, 1.570796, 1.687215],accel_mss,speed_ms,0,blend_radius_m)
    |   movel([0.116441, -1.347370, -2.593400, -0.771619, 1.570796, 1.687238],accel_mss,speed_ms,0,blend_radius_m)
    |   movel([0.116544, -1.347537, -2.593291, -0.771562, 1.570796, 1.687340],accel_mss,speed_ms,0,blend_radius_m)
    |   movel([0.117057, -1.347533, -2.593293, -0.771563, 1.570796, 1.687853],accel_mss,speed_ms,0,blend_radius_m)
    |   movel([0.117373, -1.347465, -2.593337, -0.771586, 1.570796, 1.688169],accel_mss,speed_ms,0,blend_radius_m)
    |   movel([0.117594, -1.347568, -2.593270, -0.771551, 1.570796, 1.688390],accel_mss,speed_ms,0,blend_radius_m)
    |   movel([0.117342, -1.347828, -2.593098, -0.771463, 1.570796, 1.688138],accel_mss,speed_ms,0,blend_radius_m)
    |   movel([0.117058, -1.347954, -2.593015, -0.771420, 1.570796, 1.687854],accel_mss,speed_ms,0,blend_radius_m)
    |   movel([0.116674, -1.348120, -2.592906, -0.771363, 1.570796, 1.687470],accel_mss,speed_ms,0,blend_radius_m)
    |   movel([0.116280, -1.348525, -2.592638, -0.771226, 1.570796, 1.687077],accel_mss,speed_ms,0,blend_radius_m)
    |   movel([0.116173, -1.348860, -2.592416, -0.771112, 1.570796, 1.686970],accel_mss,speed_ms,0,blend_radius_m)
    |   movel([0.116055, -1.349207, -2.592187, -0.770995, 1.570796, 1.686851],accel_mss,speed_ms,0,blend_radius_m)
    |   speed_ms = 0.003
    |   movel([0.115883, -1.352732, -2.593625, -0.766032, 1.570796, 1.686679],accel_mss,speed_ms,0,blend_radius_m)
    |   speed_ms = 0.007
    |   movel([0.115699, -1.352390, -2.593853, -0.766147, 1.570796, 1.686495],accel_mss,speed_ms,0,blend_radius_m)
    |   movel([0.115676, -1.352075, -2.594062, -0.766252, 1.570796, 1.686472],accel_mss,speed_ms,0,blend_radius_m)
    |   movel([0.115575, -1.351910, -2.594171, -0.766307, 1.570796, 1.686372],accel_mss,speed_ms,0,blend_radius_m)
    |   movel([0.115017, -1.351904, -2.594176, -0.766310, 1.570796, 1.685813],accel_mss,speed_ms,0,blend_radius_m)
    |   movel([0.114668, -1.351937, -2.594154, -0.766299, 1.570796, 1.685464],accel_mss,speed_ms,0,blend_radius_m)
    |   movel([0.114704, -1.351664, -2.594335, -0.766390, 1.570796, 1.685500],accel_mss,speed_ms,0,blend_radius_m)
    |   movel([0.115071, -1.351494, -2.594447, -0.766447, 1.570796, 1.685867],accel_mss,speed_ms,0,blend_radius_m)
    |   movel([0.115442, -1.351335, -2.594553, -0.766501, 1.570796, 1.686238],accel_mss,speed_ms,0,blend_radius_m)
    |   movel([0.115828, -1.350923, -2.594826, -0.766640, 1.570796, 1.686625],accel_mss,speed_ms,0,blend_radius_m)
    |   movel([0.115940, -1.350569, -2.595061, -0.766759, 1.570796, 1.686737],accel_mss,speed_ms,0,blend_radius_m)
    |   movel([0.116063, -1.350247, -2.595274, -0.766868, 1.570796, 1.686859],accel_mss,speed_ms,0,blend_radius_m)
    |   movel([0.116375, -1.350159, -2.595333, -0.766898, 1.570796, 1.687171],accel_mss,speed_ms,0,blend_radius_m)
    |   movel([0.116418, -1.350434, -2.595150, -0.766805, 1.570796, 1.687215],accel_mss,speed_ms,0,blend_radius_m)
    |   movel([0.116441, -1.350750, -2.594941, -0.766698, 1.570796, 1.687238],accel_mss,speed_ms,0,blend_radius_m)
    |   movel([0.116544, -1.350916, -2.594831, -0.766642, 1.570796, 1.687340],accel_mss,speed_ms,0,blend_radius_m)
    |   movel([0.117057, -1.350912, -2.594833, -0.766643, 1.570796, 1.687853],accel_mss,speed_ms,0,blend_radius_m)
    |   movel([0.117373, -1.350845, -2.594878, -0.766666, 1.570796, 1.688169],accel_mss,speed_ms,0,blend_radius_m)
    |   movel([0.117594, -1.350948, -2.594810, -0.766631, 1.570796, 1.688390],accel_mss,speed_ms,0,blend_radius_m)
    |   movel([0.117342, -1.351207, -2.594638, -0.766544, 1.570796, 1.688138],accel_mss,speed_ms,0,blend_radius_m)
    |   movel([0.117058, -1.351333, -2.594555, -0.766501, 1.570796, 1.687854],accel_mss,speed_ms,0,blend_radius_m)
    |   movel([0.116674, -1.351498, -2.594445, -0.766446, 1.570796, 1.687470],accel_mss,speed_ms,0,blend_radius_m)
    |   movel([0.116280, -1.351902, -2.594177, -0.766310, 1.570796, 1.687077],accel_mss,speed_ms,0,blend_radius_m)
    |   movel([0.116173, -1.352237, -2.593954, -0.766198, 1.570796, 1.686970],accel_mss,speed_ms,0,blend_radius_m)
    |   movel([0.116055, -1.352583, -2.593724, -0.766082, 1.570796, 1.686851],accel_mss,speed_ms,0,blend_radius_m)
    |   speed_ms = 0.003
    |   movel([0.115883, -1.339378, -2.587426, -0.785585, 1.570796, 1.686679],accel_mss,speed_ms,0,blend_radius_m)
    |   speed_ms = 1.000
    |   movel([0.115883, -1.313834, -2.574634, -0.823920, 1.570796, 1.686679],accel_mss,speed_ms,0,blend_radius_m)
    |   movel([0.116165, -1.307823, -2.578390, -0.826176, 1.570796, 1.686961],accel_mss,speed_ms,0,blend_radius_m)
    |   movel([0.116165, -1.333465, -2.591259, -0.787665, 1.570796, 1.686961],accel_mss,speed_ms,0,blend_radius_m)
    |   speed_ms = 0.003
    |   movel([0.116165, -1.343486, -2.595951, -0.772952, 1.570796, 1.686961],accel_mss,speed_ms,0,blend_radius_m)
    |   speed_ms = 0.007
    |   movel([0.115451, -1.343685, -2.595821, -0.772883, 1.570796, 1.686247],accel_mss,speed_ms,0,blend_radius_m)
    |   movel([0.115104, -1.343689, -2.595818, -0.772882, 1.570796, 1.685900],accel_mss,speed_ms,0,blend_radius_m)
    |   movel([0.115268, -1.343302, -2.596071, -0.773016, 1.570796, 1.686064],accel_mss,speed_ms,0,blend_radius_m)
    |   movel([0.115501, -1.343098, -2.596204, -0.773087, 1.570796, 1.686297],accel_mss,speed_ms,0,blend_radius_m)
    |   movel([0.115888, -1.342901, -2.596333, -0.773155, 1.570796, 1.686685],accel_mss,speed_ms,0,blend_radius_m)
    |   movel([0.116623, -1.342625, -2.596513, -0.773251, 1.570796, 1.687420],accel_mss,speed_ms,0,blend_radius_m)
    |   movel([0.117131, -1.342452, -2.596626, -0.773311, 1.570796, 1.687928],accel_mss,speed_ms,0,blend_radius_m)
    |   movel([0.117489, -1.342352, -2.596691, -0.773346, 1.570796, 1.688285],accel_mss,speed_ms,0,blend_radius_m)
    |   movel([0.117872, -1.342327, -2.596707, -0.773354, 1.570796, 1.688668],accel_mss,speed_ms,0,blend_radius_m)
    |   movel([0.118205, -1.342164, -2.596814, -0.773411, 1.570796, 1.689001],accel_mss,speed_ms,0,blend_radius_m)
    |   movel([0.118288, -1.342353, -2.596691, -0.773345, 1.570796, 1.689084],accel_mss,speed_ms,0,blend_radius_m)
    |   movel([0.117936, -1.342765, -2.596422, -0.773202, 1.570796, 1.688732],accel_mss,speed_ms,0,blend_radius_m)
    |   movel([0.117499, -1.343009, -2.596262, -0.773117, 1.570796, 1.688295],accel_mss,speed_ms,0,blend_radius_m)
    |   movel([0.116912, -1.343249, -2.596106, -0.773034, 1.570796, 1.687708],accel_mss,speed_ms,0,blend_radius_m)
    |   movel([0.116165, -1.343486, -2.595951, -0.772952, 1.570796, 1.686961],accel_mss,speed_ms,0,blend_radius_m)
    |   speed_ms = 0.003
    |   movel([0.116165, -1.346876, -2.597498, -0.768015, 1.570796, 1.686961],accel_mss,speed_ms,0,blend_radius_m)
    |   speed_ms = 0.007
    |   movel([0.115451, -1.347074, -2.597367, -0.767947, 1.570796, 1.686247],accel_mss,speed_ms,0,blend_radius_m)
    |   movel([0.115104, -1.347078, -2.597365, -0.767946, 1.570796, 1.685900],accel_mss,speed_ms,0,blend_radius_m)
    |   movel([0.115268, -1.346692, -2.597619, -0.768078, 1.570796, 1.686064],accel_mss,speed_ms,0,blend_radius_m)
    |   movel([0.115501, -1.346489, -2.597752, -0.768148, 1.570796, 1.686297],accel_mss,speed_ms,0,blend_radius_m)
    |   movel([0.115888, -1.346292, -2.597881, -0.768215, 1.570796, 1.686685],accel_mss,speed_ms,0,blend_radius_m)
    |   movel([0.116623, -1.346017, -2.598062, -0.768310, 1.570796, 1.687420],accel_mss,speed_ms,0,blend_radius_m)
    |   movel([0.117131, -1.345844, -2.598175, -0.768370, 1.570796, 1.687928],accel_mss,speed_ms,0,blend_radius_m)
    |   movel([0.117489, -1.345745, -2.598240, -0.768404, 1.570796, 1.688285],accel_mss,speed_ms,0,blend_radius_m)
    |   movel([0.117872, -1.345720, -2.598256, -0.768412, 1.570796, 1.688668],accel_mss,speed_ms,0,blend_radius_m)
    |   movel([0.118205, -1.345557, -2.598363, -0.768468, 1.570796, 1.689001],accel_mss,speed_ms,0,blend_radius_m)
    |   movel([0.118288, -1.345746, -2.598240, -0.768403, 1.570796, 1.689084],accel_mss,speed_ms,0,blend_radius_m)
    |   movel([0.117936, -1.346157, -2.597970, -0.768262, 1.570796, 1.688732],accel_mss,speed_ms,0,blend_radius_m)
    |   movel([0.117499, -1.346400, -2.597810, -0.768178, 1.570796, 1.688295],accel_mss,speed_ms,0,blend_radius_m)
    |   movel([0.116912, -1.346639, -2.597653, -0.768096, 1.570796, 1.687708],accel_mss,speed_ms,0,blend_radius_m)
    |   movel([0.116165, -1.346876, -2.597498, -0.768015, 1.570796, 1.686961],accel_mss,speed_ms,0,blend_radius_m)
    |   speed_ms = 0.003
    |   movel([0.116165, -1.333465, -2.591259, -0.787665, 1.570796, 1.686961],accel_mss,speed_ms,0,blend_radius_m)
    |   speed_ms = 1.000
    |   movel([0.116165, -1.307823, -2.578390, -0.826176, 1.570796, 1.686961],accel_mss,speed_ms,0,blend_radius_m)
    |   movel([0.116275, -1.306704, -2.579085, -0.826601, 1.570796, 1.687071],accel_mss,speed_ms,0,blend_radius_m)
    |   movel([0.116275, -1.332363, -2.591968, -0.788057, 1.570796, 1.687071],accel_mss,speed_ms,0,blend_radius_m)
    |   speed_ms = 0.003
    |   movel([0.116275, -1.342392, -2.596665, -0.773332, 1.570796, 1.687071],accel_mss,speed_ms,0,blend_radius_m)
    |   speed_ms = 0.007
    |   movel([0.114992, -1.342821, -2.596385, -0.773183, 1.570796, 1.685788],accel_mss,speed_ms,0,blend_radius_m)
    |   movel([0.115029, -1.342536, -2.596571, -0.773282, 1.570796, 1.685826],accel_mss,speed_ms,0,blend_radius_m)
    |   movel([0.115135, -1.342289, -2.596733, -0.773368, 1.570796, 1.685931],accel_mss,speed_ms,0,blend_radius_m)
    |   movel([0.115455, -1.341882, -2.596998, -0.773509, 1.570796, 1.686251],accel_mss,speed_ms,0,blend_radius_m)
    |   movel([0.115812, -1.341501, -2.597246, -0.773642, 1.570796, 1.686608],accel_mss,speed_ms,0,blend_radius_m)
    |   movel([0.116087, -1.341342, -2.597350, -0.773697, 1.570796, 1.686883],accel_mss,speed_ms,0,blend_radius_m)
    |   movel([0.116501, -1.341104, -2.597505, -0.773780, 1.570796, 1.687297],accel_mss,speed_ms,0,blend_radius_m)
    |   movel([0.117092, -1.340955, -2.597601, -0.773833, 1.570796, 1.687889],accel_mss,speed_ms,0,blend_radius_m)
    |   movel([0.117675, -1.340833, -2.597681, -0.773875, 1.570796, 1.688471],accel_mss,speed_ms,0,blend_radius_m)
    |   movel([0.117918, -1.340842, -2.597675, -0.773872, 1.570796, 1.688714],accel_mss,speed_ms,0,blend_radius_m)
    |   movel([0.118172, -1.340876, -2.597653, -0.773860, 1.570796, 1.688969],accel_mss,speed_ms,0,blend_radius_m)
    |   movel([0.118369, -1.340949, -2.597606, -0.773835, 1.570796, 1.689165],accel_mss,speed_ms,0,blend_radius_m)
    |   movel([0.118272, -1.341334, -2.597355, -0.773700, 1.570796, 1.689068],accel_mss,speed_ms,0,blend_radius_m)
    |   movel([0.118052, -1.341618, -2.597170, -0.773601, 1.570796, 1.688849],accel_mss,speed_ms,0,blend_radius_m)
    |   movel([0.117694, -1.341850, -2.597018, -0.773520, 1.570796, 1.688491],accel_mss,speed_ms,0,blend_radius_m)
    |   movel([0.117282, -1.342023, -2.596906, -0.773460, 1.570796, 1.688078],accel_mss,speed_ms,0,blend_radius_m)
    |   movel([0.116789, -1.342212, -2.596782, -0.773394, 1.570796, 1.687585],accel_mss,speed_ms,0,blend_radius_m)
    |   movel([0.116275, -1.342392, -2.596665, -0.773332, 1.570796, 1.687071],accel_mss,speed_ms,0,blend_radius_m)
    |   speed_ms = 0.003
    |   movel([0.116275, -1.345785, -2.598214, -0.768390, 1.570796, 1.687071],accel_mss,speed_ms,0,blend_radius_m)
    |   speed_ms = 0.007
    |   movel([0.114992, -1.346213, -2.597934, -0.768243, 1.570796, 1.685788],accel_mss,speed_ms,0,blend_radius_m)
    |   movel([0.115029, -1.345928, -2.598120, -0.768341, 1.570796, 1.685826],accel_mss,speed_ms,0,blend_radius_m)
    |   movel([0.115135, -1.345682, -2.598282, -0.768426, 1.570796, 1.685931],accel_mss,speed_ms,0,blend_radius_m)
    |   movel([0.115455, -1.345276, -2.598547, -0.768565, 1.570796, 1.686251],accel_mss,speed_ms,0,blend_radius_m)
    |   movel([0.115812, -1.344896, -2.598797, -0.768697, 1.570796, 1.686608],accel_mss,speed_ms,0,blend_radius_m)
    |   movel([0.116087, -1.344738, -2.598900, -0.768751, 1.570796, 1.686883],accel_mss,speed_ms,0,blend_radius_m)
    |   movel([0.116501, -1.344500, -2.599056, -0.768833, 1.570796, 1.687297],accel_mss,speed_ms,0,blend_radius_m)
    |   movel([0.117092, -1.344351, -2.599153, -0.768885, 1.570796, 1.687889],accel_mss,speed_ms,0,blend_radius_m)
    |   movel([0.117675, -1.344230, -2.599232, -0.768927, 1.570796, 1.688471],accel_mss,speed_ms,0,blend_radius_m)
    |   movel([0.117918, -1.344238, -2.599227, -0.768924, 1.570796, 1.688714],accel_mss,speed_ms,0,blend_radius_m)
    |   movel([0.118172, -1.344272, -2.599204, -0.768912, 1.570796, 1.688969],accel_mss,speed_ms,0,blend_radius_m)
    |   movel([0.118369, -1.344345, -2.599157, -0.768887, 1.570796, 1.689165],accel_mss,speed_ms,0,blend_radius_m)
    |   movel([0.118272, -1.344729, -2.598906, -0.768754, 1.570796, 1.689068],accel_mss,speed_ms,0,blend_radius_m)
    |   movel([0.118052, -1.345012, -2.598720, -0.768656, 1.570796, 1.688849],accel_mss,speed_ms,0,blend_radius_m)
    |   movel([0.117694, -1.345244, -2.598568, -0.768576, 1.570796, 1.688491],accel_mss,speed_ms,0,blend_radius_m)
    |   movel([0.117282, -1.345417, -2.598455, -0.768517, 1.570796, 1.688078],accel_mss,speed_ms,0,blend_radius_m)
    |   movel([0.116789, -1.345606, -2.598332, -0.768452, 1.570796, 1.687585],accel_mss,speed_ms,0,blend_radius_m)
    |   movel([0.116275, -1.345785, -2.598214, -0.768390, 1.570796, 1.687071],accel_mss,speed_ms,0,blend_radius_m)
    |   speed_ms = 0.003
    |   movel([0.116275, -1.332363, -2.591968, -0.788057, 1.570796, 1.687071],accel_mss,speed_ms,0,blend_radius_m)
    |   speed_ms = 1.000
    |   movel([0.116275, -1.306704, -2.579085, -0.826601, 1.570796, 1.687071],accel_mss,speed_ms,0,blend_radius_m)
    |   movel([0.110311, -1.309407, -2.577405, -0.825577, 1.570796, 1.681108],accel_mss,speed_ms,0,blend_radius_m)
    |   movel([0.110311, -1.335023, -2.590253, -0.787112, 1.570796, 1.681108],accel_mss,speed_ms,0,blend_radius_m)
    |   speed_ms = 0.003
    |   movel([0.110311, -1.345033, -2.594937, -0.772418, 1.570796, 1.681108],accel_mss,speed_ms,0,blend_radius_m)
    |   speed_ms = 0.007
    |   movel([0.110218, -1.345333, -2.594740, -0.772315, 1.570796, 1.681015],accel_mss,speed_ms,0,blend_radius_m)
    |   movel([0.110038, -1.345690, -2.594506, -0.772193, 1.570796, 1.680834],accel_mss,speed_ms,0,blend_radius_m)
    |   movel([0.109560, -1.346240, -2.594145, -0.772005, 1.570796, 1.680356],accel_mss,speed_ms,0,blend_radius_m)
    |   movel([0.108920, -1.346642, -2.593880, -0.771867, 1.570796, 1.679717],accel_mss,speed_ms,0,blend_radius_m)
    |   movel([0.108265, -1.346808, -2.593771, -0.771810, 1.570796, 1.679062],accel_mss,speed_ms,0,blend_radius_m)
    |   movel([0.107740, -1.346699, -2.593843, -0.771848, 1.570796, 1.678536],accel_mss,speed_ms,0,blend_radius_m)
    |   movel([0.107409, -1.346368, -2.594060, -0.771961, 1.570796, 1.678205],accel_mss,speed_ms,0,blend_radius_m)
    |   movel([0.107327, -1.345934, -2.594346, -0.772109, 1.570796, 1.678123],accel_mss,speed_ms,0,blend_radius_m)
    |   movel([0.107509, -1.345417, -2.594686, -0.772287, 1.570796, 1.678305],accel_mss,speed_ms,0,blend_radius_m)
    |   movel([0.107937, -1.344853, -2.595055, -0.772480, 1.570796, 1.678734],accel_mss,speed_ms,0,blend_radius_m)
    |   movel([0.108340, -1.344485, -2.595297, -0.772607, 1.570796, 1.679136],accel_mss,speed_ms,0,blend_radius_m)
    |   movel([0.108727, -1.344242, -2.595456, -0.772691, 1.570796, 1.679523],accel_mss,speed_ms,0,blend_radius_m)
    |   movel([0.109109, -1.344122, -2.595535, -0.772732, 1.570796, 1.679905],accel_mss,speed_ms,0,blend_radius_m)
    |   movel([0.109499, -1.344117, -2.595538, -0.772734, 1.570796, 1.680296],accel_mss,speed_ms,0,blend_radius_m)
    |   movel([0.109823, -1.344224, -2.595468, -0.772697, 1.570796, 1.680619],accel_mss,speed_ms,0,blend_radius_m)
    |   movel([0.110099, -1.344446, -2.595322, -0.772621, 1.570796, 1.680895],accel_mss,speed_ms,0,blend_radius_m)
    |   movel([0.110276, -1.344735, -2.595133, -0.772521, 1.570796, 1.681072],accel_mss,speed_ms,0,blend_radius_m)
    |   movel([0.110311, -1.345033, -2.594937, -0.772418, 1.570796, 1.681108],accel_mss,speed_ms,0,blend_radius_m)
    |   speed_ms = 0.003
    |   movel([0.110311, -1.348419, -2.596482, -0.767488, 1.570796, 1.681108],accel_mss,speed_ms,0,blend_radius_m)
    |   speed_ms = 0.007
    |   movel([0.110218, -1.348719, -2.596284, -0.767386, 1.570796, 1.681015],accel_mss,speed_ms,0,blend_radius_m)
    |   movel([0.110038, -1.349074, -2.596050, -0.767265, 1.570796, 1.680834],accel_mss,speed_ms,0,blend_radius_m)
    |   movel([0.109560, -1.349623, -2.595687, -0.767079, 1.570796, 1.680356],accel_mss,speed_ms,0,blend_radius_m)
    |   movel([0.108920, -1.350024, -2.595422, -0.766943, 1.570796, 1.679717],accel_mss,speed_ms,0,blend_radius_m)
    |   movel([0.108265, -1.350189, -2.595312, -0.766887, 1.570796, 1.679062],accel_mss,speed_ms,0,blend_radius_m)
    |   movel([0.107740, -1.350080, -2.595384, -0.766924, 1.570796, 1.678536],accel_mss,speed_ms,0,blend_radius_m)
    |   movel([0.107409, -1.349751, -2.595603, -0.767036, 1.570796, 1.678205],accel_mss,speed_ms,0,blend_radius_m)
    |   movel([0.107327, -1.349318, -2.595889, -0.767182, 1.570796, 1.678123],accel_mss,speed_ms,0,blend_radius_m)
    |   movel([0.107509, -1.348802, -2.596229, -0.767358, 1.570796, 1.678305],accel_mss,speed_ms,0,blend_radius_m)
    |   movel([0.107937, -1.348240, -2.596600, -0.767549, 1.570796, 1.678734],accel_mss,speed_ms,0,blend_radius_m)
    |   movel([0.108340, -1.347872, -2.596842, -0.767675, 1.570796, 1.679136],accel_mss,speed_ms,0,blend_radius_m)
    |   movel([0.108727, -1.347630, -2.597002, -0.767757, 1.570796, 1.679523],accel_mss,speed_ms,0,blend_radius_m)
    |   movel([0.109109, -1.347510, -2.597081, -0.767798, 1.570796, 1.679905],accel_mss,speed_ms,0,blend_radius_m)
    |   movel([0.109499, -1.347505, -2.597084, -0.767800, 1.570796, 1.680296],accel_mss,speed_ms,0,blend_radius_m)
    |   movel([0.109823, -1.347612, -2.597014, -0.767763, 1.570796, 1.680619],accel_mss,speed_ms,0,blend_radius_m)
    |   movel([0.110099, -1.347834, -2.596868, -0.767688, 1.570796, 1.680895],accel_mss,speed_ms,0,blend_radius_m)
    |   movel([0.110276, -1.348121, -2.596678, -0.767589, 1.570796, 1.681072],accel_mss,speed_ms,0,blend_radius_m)
    |   movel([0.110311, -1.348419, -2.596482, -0.767488, 1.570796, 1.681108],accel_mss,speed_ms,0,blend_radius_m)
    |   speed_ms = 0.003
    |   movel([0.110311, -1.335023, -2.590253, -0.787112, 1.570796, 1.681108],accel_mss,speed_ms,0,blend_radius_m)
    |   speed_ms = 1.000
    |   movel([0.110311, -1.309407, -2.577405, -0.825577, 1.570796, 1.681108],accel_mss,speed_ms,0,blend_radius_m)
    |   movel([0.104721, -1.314744, -2.574062, -0.823583, 1.570796, 1.675517],accel_mss,speed_ms,0,blend_radius_m)
    |   movel([0.104721, -1.340273, -2.586841, -0.785274, 1.570796, 1.675517],accel_mss,speed_ms,0,blend_radius_m)
    |   speed_ms = 0.003
    |   movel([0.104721, -1.350245, -2.591499, -0.770645, 1.570796, 1.675517],accel_mss,speed_ms,0,blend_radius_m)
    |   speed_ms = 0.007
    |   movel([0.104431, -1.350657, -2.591226, -0.770506, 1.570796, 1.675228],accel_mss,speed_ms,0,blend_radius_m)
    |   movel([0.104261, -1.350893, -2.591069, -0.770427, 1.570796, 1.675057],accel_mss,speed_ms,0,blend_radius_m)
    |   movel([0.103928, -1.351335, -2.590776, -0.770279, 1.570796, 1.674724],accel_mss,speed_ms,0,blend_radius_m)
    |   movel([0.103535, -1.351849, -2.590434, -0.770106, 1.570796, 1.674331],accel_mss,speed_ms,0,blend_radius_m)
    |   movel([0.103125, -1.352380, -2.590080, -0.769929, 1.570796, 1.673921],accel_mss,speed_ms,0,blend_radius_m)
    |   movel([0.102659, -1.352967, -2.589688, -0.769733, 1.570796, 1.673455],accel_mss,speed_ms,0,blend_radius_m)
    |   movel([0.102306, -1.353375, -2.589417, -0.769598, 1.570796, 1.673103],accel_mss,speed_ms,0,blend_radius_m)
    |   movel([0.102040, -1.353644, -2.589237, -0.769508, 1.570796, 1.672837],accel_mss,speed_ms,0,blend_radius_m)
    |   movel([0.101752, -1.353700, -2.589200, -0.769490, 1.570796, 1.672548],accel_mss,speed_ms,0,blend_radius_m)
    |   movel([0.101801, -1.353407, -2.589395, -0.769587, 1.570796, 1.672598],accel_mss,speed_ms,0,blend_radius_m)
    |   movel([0.102838, -1.352207, -2.590195, -0.769987, 1.570796, 1.673635],accel_mss,speed_ms,0,blend_radius_m)
    |   movel([0.103828, -1.351089, -2.590939, -0.770361, 1.570796, 1.674624],accel_mss,speed_ms,0,blend_radius_m)
    |   movel([0.104352, -1.350571, -2.591283, -0.770535, 1.570796, 1.675148],accel_mss,speed_ms,0,blend_radius_m)
    |   movel([0.104721, -1.350245, -2.591499, -0.770645, 1.570796, 1.675517],accel_mss,speed_ms,0,blend_radius_m)
    |   speed_ms = 0.003
    |   movel([0.104721, -1.353618, -2.593035, -0.765736, 1.570796, 1.675517],accel_mss,speed_ms,0,blend_radius_m)
    |   speed_ms = 0.007
    |   movel([0.104431, -1.354029, -2.592761, -0.765599, 1.570796, 1.675228],accel_mss,speed_ms,0,blend_radius_m)
    |   movel([0.104261, -1.354264, -2.592604, -0.765521, 1.570796, 1.675057],accel_mss,speed_ms,0,blend_radius_m)
    |   movel([0.103928, -1.354705, -2.592310, -0.765375, 1.570796, 1.674724],accel_mss,speed_ms,0,blend_radius_m)
    |   movel([0.103535, -1.355217, -2.591967, -0.765205, 1.570796, 1.674331],accel_mss,speed_ms,0,blend_radius_m)
    |   movel([0.103125, -1.355748, -2.591612, -0.765029, 1.570796, 1.673921],accel_mss,speed_ms,0,blend_radius_m)
    |   movel([0.102659, -1.356333, -2.591220, -0.764836, 1.570796, 1.673455],accel_mss,speed_ms,0,blend_radius_m)
    |   movel([0.102306, -1.356740, -2.590947, -0.764702, 1.570796, 1.673103],accel_mss,speed_ms,0,blend_radius_m)
    |   movel([0.102040, -1.357008, -2.590767, -0.764614, 1.570796, 1.672837],accel_mss,speed_ms,0,blend_radius_m)
    |   movel([0.101752, -1.357064, -2.590730, -0.764596, 1.570796, 1.672548],accel_mss,speed_ms,0,blend_radius_m)
    |   movel([0.101801, -1.356771, -2.590926, -0.764692, 1.570796, 1.672598],accel_mss,speed_ms,0,blend_radius_m)
    |   movel([0.102838, -1.355574, -2.591728, -0.765087, 1.570796, 1.673635],accel_mss,speed_ms,0,blend_radius_m)
    |   movel([0.103828, -1.354460, -2.592473, -0.765456, 1.570796, 1.674624],accel_mss,speed_ms,0,blend_radius_m)
    |   movel([0.104352, -1.353943, -2.592818, -0.765628, 1.570796, 1.675148],accel_mss,speed_ms,0,blend_radius_m)
    |   movel([0.104721, -1.353618, -2.593035, -0.765736, 1.570796, 1.675517],accel_mss,speed_ms,0,blend_radius_m)
    |   speed_ms = 0.003
    |   movel([0.104721, -1.340273, -2.586841, -0.785274, 1.570796, 1.675517],accel_mss,speed_ms,0,blend_radius_m)
    |   speed_ms = 1.000
    |   movel([0.104721, -1.314744, -2.574062, -0.823583, 1.570796, 1.675517],accel_mss,speed_ms,0,blend_radius_m)
    |   movel([0.129209, -1.310300, -2.576848, -0.825241, 1.570796, 1.700005],accel_mss,speed_ms,0,blend_radius_m)
    |   movel([0.129209, -1.335902, -2.589685, -0.786802, 1.570796, 1.700005],accel_mss,speed_ms,0,blend_radius_m)
    |   speed_ms = 0.003
    |   movel([0.129209, -1.345905, -2.594365, -0.772119, 1.570796, 1.700005],accel_mss,speed_ms,0,blend_radius_m)
    |   speed_ms = 0.007
    |   movel([0.130130, -1.345778, -2.594448, -0.772163, 1.570796, 1.700926],accel_mss,speed_ms,0,blend_radius_m)
    |   movel([0.130918, -1.345778, -2.594448, -0.772163, 1.570796, 1.701714],accel_mss,speed_ms,0,blend_radius_m)
    |   movel([0.131621, -1.345811, -2.594427, -0.772151, 1.570796, 1.702417],accel_mss,speed_ms,0,blend_radius_m)
    |   movel([0.131927, -1.345942, -2.594340, -0.772106, 1.570796, 1.702724],accel_mss,speed_ms,0,blend_radius_m)
    |   movel([0.131753, -1.346175, -2.594188, -0.772027, 1.570796, 1.702549],accel_mss,speed_ms,0,blend_radius_m)
    |   movel([0.131438, -1.346266, -2.594127, -0.771995, 1.570796, 1.702234],accel_mss,speed_ms,0,blend_radius_m)
    |   movel([0.130444, -1.346251, -2.594137, -0.772001, 1.570796, 1.701240],accel_mss,speed_ms,0,blend_radius_m)
    |   movel([0.129464, -1.346204, -2.594168, -0.772017, 1.570796, 1.700260],accel_mss,speed_ms,0,blend_radius_m)
    |   movel([0.129246, -1.346094, -2.594241, -0.772055, 1.570796, 1.700042],accel_mss,speed_ms,0,blend_radius_m)
    |   speed_ms = 0.003
    |   movel([0.129209, -1.349289, -2.595908, -0.767192, 1.570796, 1.700005],accel_mss,speed_ms,0,blend_radius_m)
    |   speed_ms = 0.007
    |   movel([0.130130, -1.349162, -2.595992, -0.767235, 1.570796, 1.700926],accel_mss,speed_ms,0,blend_radius_m)
    |   movel([0.130918, -1.349162, -2.595991, -0.767235, 1.570796, 1.701714],accel_mss,speed_ms,0,blend_radius_m)
    |   movel([0.131621, -1.349195, -2.595970, -0.767224, 1.570796, 1.702417],accel_mss,speed_ms,0,blend_radius_m)
    |   movel([0.131927, -1.349326, -2.595883, -0.767180, 1.570796, 1.702724],accel_mss,speed_ms,0,blend_radius_m)
    |   movel([0.131753, -1.349558, -2.595730, -0.767101, 1.570796, 1.702549],accel_mss,speed_ms,0,blend_radius_m)
    |   movel([0.131438, -1.349649, -2.595670, -0.767070, 1.570796, 1.702234],accel_mss,speed_ms,0,blend_radius_m)
    |   movel([0.130444, -1.349634, -2.595680, -0.767075, 1.570796, 1.701240],accel_mss,speed_ms,0,blend_radius_m)
    |   movel([0.129464, -1.349587, -2.595711, -0.767091, 1.570796, 1.700260],accel_mss,speed_ms,0,blend_radius_m)
    |   movel([0.129246, -1.349477, -2.595784, -0.767128, 1.570796, 1.700042],accel_mss,speed_ms,0,blend_radius_m)
    |   speed_ms = 0.003
    |   movel([0.129209, -1.335902, -2.589685, -0.786802, 1.570796, 1.700005],accel_mss,speed_ms,0,blend_radius_m)
    |   speed_ms = 1.000
    |   movel([0.129209, -1.310300, -2.576848, -0.825241, 1.570796, 1.700005],accel_mss,speed_ms,0,blend_radius_m)
    |   movel([0.133372, -1.307920, -2.578330, -0.826139, 1.570796, 1.704169],accel_mss,speed_ms,0,blend_radius_m)
    |   movel([0.133372, -1.333561, -2.591198, -0.787631, 1.570796, 1.704169],accel_mss,speed_ms,0,blend_radius_m)
    |   speed_ms = 0.003
    |   movel([0.133372, -1.343581, -2.595889, -0.772919, 1.570796, 1.704169],accel_mss,speed_ms,0,blend_radius_m)
    |   speed_ms = 0.007
    |   movel([0.133523, -1.343804, -2.595743, -0.772842, 1.570796, 1.704320],accel_mss,speed_ms,0,blend_radius_m)
    |   movel([0.133757, -1.343909, -2.595674, -0.772806, 1.570796, 1.704553],accel_mss,speed_ms,0,blend_radius_m)
    |   movel([0.133786, -1.344214, -2.595475, -0.772701, 1.570796, 1.704582],accel_mss,speed_ms,0,blend_radius_m)
    |   movel([0.133733, -1.344526, -2.595270, -0.772593, 1.570796, 1.704530],accel_mss,speed_ms,0,blend_radius_m)
    |   movel([0.133693, -1.344774, -2.595107, -0.772508, 1.570796, 1.704490],accel_mss,speed_ms,0,blend_radius_m)
    |   movel([0.133685, -1.345123, -2.594878, -0.772387, 1.570796, 1.704481],accel_mss,speed_ms,0,blend_radius_m)
    |   movel([0.133764, -1.345308, -2.594757, -0.772324, 1.570796, 1.704561],accel_mss,speed_ms,0,blend_radius_m)
    |   movel([0.133678, -1.345762, -2.594459, -0.772168, 1.570796, 1.704474],accel_mss,speed_ms,0,blend_radius_m)
    |   movel([0.133620, -1.346014, -2.594293, -0.772082, 1.570796, 1.704416],accel_mss,speed_ms,0,blend_radius_m)
    |   movel([0.133584, -1.346401, -2.594039, -0.771949, 1.570796, 1.704380],accel_mss,speed_ms,0,blend_radius_m)
    |   movel([0.133696, -1.346576, -2.593924, -0.771890, 1.570796, 1.704493],accel_mss,speed_ms,0,blend_radius_m)
    |   movel([0.133614, -1.347215, -2.593502, -0.771671, 1.570796, 1.704411],accel_mss,speed_ms,0,blend_radius_m)
    |   movel([0.133501, -1.347865, -2.593074, -0.771450, 1.570796, 1.704297],accel_mss,speed_ms,0,blend_radius_m)
    |   movel([0.133318, -1.348123, -2.592904, -0.771362, 1.570796, 1.704114],accel_mss,speed_ms,0,blend_radius_m)
    |   movel([0.133224, -1.348613, -2.592580, -0.771196, 1.570796, 1.704020],accel_mss,speed_ms,0,blend_radius_m)
    |   movel([0.133196, -1.348926, -2.592373, -0.771090, 1.570796, 1.703993],accel_mss,speed_ms,0,blend_radius_m)
    |   movel([0.133171, -1.349242, -2.592164, -0.770983, 1.570796, 1.703967],accel_mss,speed_ms,0,blend_radius_m)
    |   movel([0.133130, -1.349497, -2.591995, -0.770897, 1.570796, 1.703926],accel_mss,speed_ms,0,blend_radius_m)
    |   movel([0.133029, -1.349737, -2.591836, -0.770816, 1.570796, 1.703825],accel_mss,speed_ms,0,blend_radius_m)
    |   movel([0.132912, -1.350001, -2.591661, -0.770727, 1.570796, 1.703709],accel_mss,speed_ms,0,blend_radius_m)
    |   movel([0.132787, -1.350833, -2.591109, -0.770447, 1.570796, 1.703583],accel_mss,speed_ms,0,blend_radius_m)
    |   movel([0.132241, -1.352571, -2.589953, -0.769865, 1.570796, 1.703037],accel_mss,speed_ms,0,blend_radius_m)
    |   movel([0.131630, -1.354418, -2.588720, -0.769252, 1.570796, 1.702426],accel_mss,speed_ms,0,blend_radius_m)
    |   movel([0.131422, -1.354684, -2.588541, -0.769163, 1.570796, 1.702219],accel_mss,speed_ms,0,blend_radius_m)
    |   movel([0.131217, -1.355020, -2.588316, -0.769053, 1.570796, 1.702013],accel_mss,speed_ms,0,blend_radius_m)
    |   movel([0.131469, -1.355313, -2.588120, -0.768956, 1.570796, 1.702265],accel_mss,speed_ms,0,blend_radius_m)
    |   movel([0.131675, -1.355437, -2.588037, -0.768915, 1.570796, 1.702471],accel_mss,speed_ms,0,blend_radius_m)
    |   movel([0.131656, -1.355707, -2.587856, -0.768826, 1.570796, 1.702453],accel_mss,speed_ms,0,blend_radius_m)
    |   movel([0.131428, -1.355961, -2.587685, -0.768742, 1.570796, 1.702225],accel_mss,speed_ms,0,blend_radius_m)
    |   movel([0.131132, -1.356262, -2.587483, -0.768644, 1.570796, 1.701929],accel_mss,speed_ms,0,blend_radius_m)
    |   movel([0.127085, -1.356793, -2.587126, -0.768469, 1.570796, 1.697882],accel_mss,speed_ms,0,blend_radius_m)
    |   movel([0.125499, -1.357008, -2.586982, -0.768399, 1.570796, 1.696296],accel_mss,speed_ms,0,blend_radius_m)
    |   movel([0.124079, -1.357201, -2.586852, -0.768336, 1.570796, 1.694875],accel_mss,speed_ms,0,blend_radius_m)
    |   movel([0.122882, -1.357368, -2.586740, -0.768282, 1.570796, 1.693678],accel_mss,speed_ms,0,blend_radius_m)
    |   movel([0.122534, -1.357421, -2.586704, -0.768264, 1.570796, 1.693331],accel_mss,speed_ms,0,blend_radius_m)
    |   movel([0.122267, -1.357464, -2.586675, -0.768250, 1.570796, 1.693063],accel_mss,speed_ms,0,blend_radius_m)
    |   movel([0.121847, -1.357524, -2.586635, -0.768230, 1.570796, 1.692643],accel_mss,speed_ms,0,blend_radius_m)
    |   movel([0.121369, -1.357592, -2.586589, -0.768208, 1.570796, 1.692165],accel_mss,speed_ms,0,blend_radius_m)
    |   movel([0.120899, -1.357655, -2.586546, -0.768188, 1.570796, 1.691695],accel_mss,speed_ms,0,blend_radius_m)
    |   movel([0.120401, -1.357724, -2.586500, -0.768165, 1.570796, 1.691197],accel_mss,speed_ms,0,blend_radius_m)
    |   movel([0.119840, -1.357800, -2.586449, -0.768140, 1.570796, 1.690636],accel_mss,speed_ms,0,blend_radius_m)
    |   movel([0.119304, -1.357875, -2.586398, -0.768116, 1.570796, 1.690101],accel_mss,speed_ms,0,blend_radius_m)
    |   movel([0.118887, -1.357934, -2.586358, -0.768097, 1.570796, 1.689683],accel_mss,speed_ms,0,blend_radius_m)
    |   movel([0.118469, -1.357995, -2.586317, -0.768077, 1.570796, 1.689265],accel_mss,speed_ms,0,blend_radius_m)
    |   movel([0.117933, -1.358069, -2.586268, -0.768053, 1.570796, 1.688730],accel_mss,speed_ms,0,blend_radius_m)
    |   movel([0.117372, -1.358148, -2.586214, -0.768027, 1.570796, 1.688169],accel_mss,speed_ms,0,blend_radius_m)
    |   movel([0.116874, -1.358218, -2.586167, -0.768004, 1.570796, 1.687671],accel_mss,speed_ms,0,blend_radius_m)
    |   movel([0.114544, -1.358551, -2.585942, -0.767896, 1.570796, 1.685341],accel_mss,speed_ms,0,blend_radius_m)
    |   movel([0.111844, -1.358958, -2.585668, -0.767764, 1.570796, 1.682641],accel_mss,speed_ms,0,blend_radius_m)
    |   movel([0.109120, -1.359383, -2.585380, -0.767626, 1.570796, 1.679916],accel_mss,speed_ms,0,blend_radius_m)
    |   movel([0.108772, -1.359460, -2.585328, -0.767601, 1.570796, 1.679568],accel_mss,speed_ms,0,blend_radius_m)
    |   movel([0.108514, -1.359224, -2.585488, -0.767677, 1.570796, 1.679311],accel_mss,speed_ms,0,blend_radius_m)
    |   movel([0.108672, -1.358892, -2.585712, -0.767785, 1.570796, 1.679468],accel_mss,speed_ms,0,blend_radius_m)
    |   movel([0.108981, -1.358556, -2.585939, -0.767894, 1.570796, 1.679777],accel_mss,speed_ms,0,blend_radius_m)
    |   movel([0.109311, -1.358296, -2.586114, -0.767979, 1.570796, 1.680107],accel_mss,speed_ms,0,blend_radius_m)
    |   movel([0.109605, -1.358120, -2.586233, -0.768036, 1.570796, 1.680401],accel_mss,speed_ms,0,blend_radius_m)
    |   movel([0.109666, -1.357828, -2.586430, -0.768131, 1.570796, 1.680463],accel_mss,speed_ms,0,blend_radius_m)
    |   movel([0.109470, -1.357719, -2.586503, -0.768167, 1.570796, 1.680266],accel_mss,speed_ms,0,blend_radius_m)
    |   movel([0.109530, -1.357479, -2.586665, -0.768245, 1.570796, 1.680326],accel_mss,speed_ms,0,blend_radius_m)
    |   movel([0.109705, -1.357223, -2.586837, -0.768329, 1.570796, 1.680502],accel_mss,speed_ms,0,blend_radius_m)
    |   movel([0.109652, -1.356857, -2.587083, -0.768449, 1.570796, 1.680449],accel_mss,speed_ms,0,blend_radius_m)
    |   movel([0.109837, -1.356609, -2.587250, -0.768530, 1.570796, 1.680633],accel_mss,speed_ms,0,blend_radius_m)
    |   movel([0.109967, -1.356167, -2.587547, -0.768675, 1.570796, 1.680764],accel_mss,speed_ms,0,blend_radius_m)
    |   movel([0.110006, -1.355882, -2.587738, -0.768768, 1.570796, 1.680802],accel_mss,speed_ms,0,blend_radius_m)
    |   movel([0.110093, -1.355310, -2.588122, -0.768957, 1.570796, 1.680889],accel_mss,speed_ms,0,blend_radius_m)
    |   movel([0.110206, -1.354843, -2.588435, -0.769111, 1.570796, 1.681003],accel_mss,speed_ms,0,blend_radius_m)
    |   movel([0.110408, -1.354229, -2.588846, -0.769314, 1.570796, 1.681205],accel_mss,speed_ms,0,blend_radius_m)
    |   movel([0.110894, -1.352904, -2.589731, -0.769754, 1.570796, 1.681691],accel_mss,speed_ms,0,blend_radius_m)
    |   movel([0.111101, -1.352357, -2.590096, -0.769937, 1.570796, 1.681897],accel_mss,speed_ms,0,blend_radius_m)
    |   movel([0.111293, -1.351885, -2.590410, -0.770094, 1.570796, 1.682089],accel_mss,speed_ms,0,blend_radius_m)
    |   movel([0.111466, -1.351484, -2.590676, -0.770229, 1.570796, 1.682262],accel_mss,speed_ms,0,blend_radius_m)
    |   movel([0.111570, -1.351218, -2.590853, -0.770318, 1.570796, 1.682366],accel_mss,speed_ms,0,blend_radius_m)
    |   movel([0.111744, -1.350968, -2.591019, -0.770402, 1.570796, 1.682540],accel_mss,speed_ms,0,blend_radius_m)
    |   movel([0.111777, -1.350613, -2.591255, -0.770521, 1.570796, 1.682573],accel_mss,speed_ms,0,blend_radius_m)
    |   movel([0.112301, -1.349502, -2.591991, -0.770895, 1.570796, 1.683097],accel_mss,speed_ms,0,blend_radius_m)
    |   movel([0.112851, -1.348413, -2.592712, -0.771264, 1.570796, 1.683647],accel_mss,speed_ms,0,blend_radius_m)
    |   movel([0.113284, -1.347690, -2.593189, -0.771509, 1.570796, 1.684081],accel_mss,speed_ms,0,blend_radius_m)
    |   movel([0.113462, -1.347437, -2.593356, -0.771596, 1.570796, 1.684258],accel_mss,speed_ms,0,blend_radius_m)
    |   movel([0.113667, -1.347170, -2.593532, -0.771687, 1.570796, 1.684463],accel_mss,speed_ms,0,blend_radius_m)
    |   movel([0.113872, -1.346920, -2.593697, -0.771772, 1.570796, 1.684668],accel_mss,speed_ms,0,blend_radius_m)
    |   movel([0.114255, -1.346494, -2.593977, -0.771917, 1.570796, 1.685052],accel_mss,speed_ms,0,blend_radius_m)
    |   movel([0.114419, -1.346139, -2.594211, -0.772039, 1.570796, 1.685216],accel_mss,speed_ms,0,blend_radius_m)
    |   movel([0.114172, -1.346157, -2.594199, -0.772033, 1.570796, 1.684968],accel_mss,speed_ms,0,blend_radius_m)
    |   movel([0.113906, -1.346180, -2.594184, -0.772025, 1.570796, 1.684702],accel_mss,speed_ms,0,blend_radius_m)
    |   movel([0.113638, -1.346105, -2.594234, -0.772051, 1.570796, 1.684434],accel_mss,speed_ms,0,blend_radius_m)
    |   movel([0.113581, -1.345731, -2.594479, -0.772179, 1.570796, 1.684377],accel_mss,speed_ms,0,blend_radius_m)
    |   movel([0.113640, -1.345330, -2.594742, -0.772316, 1.570796, 1.684437],accel_mss,speed_ms,0,blend_radius_m)
    |   movel([0.113813, -1.345065, -2.594916, -0.772408, 1.570796, 1.684609],accel_mss,speed_ms,0,blend_radius_m)
    |   movel([0.114104, -1.344827, -2.595072, -0.772489, 1.570796, 1.684901],accel_mss,speed_ms,0,blend_radius_m)
    |   movel([0.114427, -1.344625, -2.595205, -0.772559, 1.570796, 1.685223],accel_mss,speed_ms,0,blend_radius_m)
    |   movel([0.114780, -1.344455, -2.595316, -0.772617, 1.570796, 1.685576],accel_mss,speed_ms,0,blend_radius_m)
    |   movel([0.115153, -1.344327, -2.595400, -0.772662, 1.570796, 1.685950],accel_mss,speed_ms,0,blend_radius_m)
    |   movel([0.115538, -1.344186, -2.595493, -0.772710, 1.570796, 1.686334],accel_mss,speed_ms,0,blend_radius_m)
    |   movel([0.116178, -1.343789, -2.595752, -0.772847, 1.570796, 1.686974],accel_mss,speed_ms,0,blend_radius_m)
    |   movel([0.118416, -1.343039, -2.596243, -0.773107, 1.570796, 1.689213],accel_mss,speed_ms,0,blend_radius_m)
    |   movel([0.120675, -1.342306, -2.596722, -0.773362, 1.570796, 1.691471],accel_mss,speed_ms,0,blend_radius_m)
    |   movel([0.120996, -1.342326, -2.596708, -0.773355, 1.570796, 1.691792],accel_mss,speed_ms,0,blend_radius_m)
    |   movel([0.121352, -1.342346, -2.596696, -0.773348, 1.570796, 1.692148],accel_mss,speed_ms,0,blend_radius_m)
    |   movel([0.121691, -1.342126, -2.596839, -0.773424, 1.570796, 1.692487],accel_mss,speed_ms,0,blend_radius_m)
    |   movel([0.121589, -1.341884, -2.596996, -0.773508, 1.570796, 1.692385],accel_mss,speed_ms,0,blend_radius_m)
    |   movel([0.121500, -1.341581, -2.597194, -0.773614, 1.570796, 1.692296],accel_mss,speed_ms,0,blend_radius_m)
    |   movel([0.121695, -1.341353, -2.597342, -0.773694, 1.570796, 1.692491],accel_mss,speed_ms,0,blend_radius_m)
    |   movel([0.122038, -1.341103, -2.597505, -0.773781, 1.570796, 1.692835],accel_mss,speed_ms,0,blend_radius_m)
    |   movel([0.122298, -1.340917, -2.597626, -0.773846, 1.570796, 1.693094],accel_mss,speed_ms,0,blend_radius_m)
    |   movel([0.122428, -1.340654, -2.597797, -0.773938, 1.570796, 1.693224],accel_mss,speed_ms,0,blend_radius_m)
    |   movel([0.122134, -1.340648, -2.597801, -0.773940, 1.570796, 1.692931],accel_mss,speed_ms,0,blend_radius_m)
    |   movel([0.121865, -1.340652, -2.597798, -0.773938, 1.570796, 1.692661],accel_mss,speed_ms,0,blend_radius_m)
    |   movel([0.121926, -1.340137, -2.598133, -0.774119, 1.570796, 1.692722],accel_mss,speed_ms,0,blend_radius_m)
    |   movel([0.122108, -1.339570, -2.598501, -0.774318, 1.570796, 1.692904],accel_mss,speed_ms,0,blend_radius_m)
    |   movel([0.122198, -1.339304, -2.598673, -0.774411, 1.570796, 1.692994],accel_mss,speed_ms,0,blend_radius_m)
    |   movel([0.122277, -1.339057, -2.598834, -0.774498, 1.570796, 1.693074],accel_mss,speed_ms,0,blend_radius_m)
    |   movel([0.122367, -1.338753, -2.599030, -0.774605, 1.570796, 1.693164],accel_mss,speed_ms,0,blend_radius_m)
    |   movel([0.122577, -1.338442, -2.599232, -0.774715, 1.570796, 1.693373],accel_mss,speed_ms,0,blend_radius_m)
    |   movel([0.122789, -1.338186, -2.599397, -0.774806, 1.570796, 1.693585],accel_mss,speed_ms,0,blend_radius_m)
    |   movel([0.123034, -1.337910, -2.599576, -0.774903, 1.570796, 1.693831],accel_mss,speed_ms,0,blend_radius_m)
    |   movel([0.123671, -1.337217, -2.600024, -0.775149, 1.570796, 1.694467],accel_mss,speed_ms,0,blend_radius_m)
    |   movel([0.124629, -1.337021, -2.600150, -0.775218, 1.570796, 1.695426],accel_mss,speed_ms,0,blend_radius_m)
    |   movel([0.125882, -1.336797, -2.600295, -0.775298, 1.570796, 1.696678],accel_mss,speed_ms,0,blend_radius_m)
    |   movel([0.127200, -1.336622, -2.600407, -0.775360, 1.570796, 1.697996],accel_mss,speed_ms,0,blend_radius_m)
    |   movel([0.128376, -1.336509, -2.600480, -0.775400, 1.570796, 1.699172],accel_mss,speed_ms,0,blend_radius_m)
    |   movel([0.128803, -1.336554, -2.600451, -0.775384, 1.570796, 1.699599],accel_mss,speed_ms,0,blend_radius_m)
    |   movel([0.129089, -1.336680, -2.600370, -0.775339, 1.570796, 1.699886],accel_mss,speed_ms,0,blend_radius_m)
    |   movel([0.129309, -1.336847, -2.600262, -0.775280, 1.570796, 1.700106],accel_mss,speed_ms,0,blend_radius_m)
    |   movel([0.129435, -1.337023, -2.600149, -0.775218, 1.570796, 1.700231],accel_mss,speed_ms,0,blend_radius_m)
    |   movel([0.129396, -1.337284, -2.599980, -0.775125, 1.570796, 1.700193],accel_mss,speed_ms,0,blend_radius_m)
    |   movel([0.129524, -1.337460, -2.599866, -0.775062, 1.570796, 1.700320],accel_mss,speed_ms,0,blend_radius_m)
    |   movel([0.129472, -1.337779, -2.599661, -0.774950, 1.570796, 1.700269],accel_mss,speed_ms,0,blend_radius_m)
    |   movel([0.129264, -1.338017, -2.599507, -0.774865, 1.570796, 1.700060],accel_mss,speed_ms,0,blend_radius_m)
    |   movel([0.129247, -1.338303, -2.599322, -0.774764, 1.570796, 1.700043],accel_mss,speed_ms,0,blend_radius_m)
    |   movel([0.129226, -1.338701, -2.599064, -0.774624, 1.570796, 1.700023],accel_mss,speed_ms,0,blend_radius_m)
    |   movel([0.129118, -1.339164, -2.598765, -0.774461, 1.570796, 1.699915],accel_mss,speed_ms,0,blend_radius_m)
    |   movel([0.128966, -1.339555, -2.598510, -0.774323, 1.570796, 1.699762],accel_mss,speed_ms,0,blend_radius_m)
    |   movel([0.128664, -1.339692, -2.598422, -0.774275, 1.570796, 1.699461],accel_mss,speed_ms,0,blend_radius_m)
    |   movel([0.128382, -1.339893, -2.598292, -0.774205, 1.570796, 1.699178],accel_mss,speed_ms,0,blend_radius_m)
    |   movel([0.128379, -1.340190, -2.598099, -0.774100, 1.570796, 1.699175],accel_mss,speed_ms,0,blend_radius_m)
    |   movel([0.128483, -1.340437, -2.597939, -0.774014, 1.570796, 1.699279],accel_mss,speed_ms,0,blend_radius_m)
    |   movel([0.128519, -1.340727, -2.597750, -0.773912, 1.570796, 1.699315],accel_mss,speed_ms,0,blend_radius_m)
    |   movel([0.128237, -1.340991, -2.597578, -0.773820, 1.570796, 1.699033],accel_mss,speed_ms,0,blend_radius_m)
    |   movel([0.128151, -1.341286, -2.597386, -0.773717, 1.570796, 1.698948],accel_mss,speed_ms,0,blend_radius_m)
    |   movel([0.128545, -1.341249, -2.597410, -0.773730, 1.570796, 1.699342],accel_mss,speed_ms,0,blend_radius_m)
    |   movel([0.129417, -1.341135, -2.597484, -0.773769, 1.570796, 1.700213],accel_mss,speed_ms,0,blend_radius_m)
    |   movel([0.130216, -1.341116, -2.597497, -0.773776, 1.570796, 1.701013],accel_mss,speed_ms,0,blend_radius_m)
    |   movel([0.130962, -1.341141, -2.597481, -0.773768, 1.570796, 1.701758],accel_mss,speed_ms,0,blend_radius_m)
    |   movel([0.131239, -1.341229, -2.597423, -0.773737, 1.570796, 1.702036],accel_mss,speed_ms,0,blend_radius_m)
    |   movel([0.131699, -1.341255, -2.597406, -0.773728, 1.570796, 1.702495],accel_mss,speed_ms,0,blend_radius_m)
    |   movel([0.132047, -1.341071, -2.597526, -0.773792, 1.570796, 1.702843],accel_mss,speed_ms,0,blend_radius_m)
    |   movel([0.131918, -1.340895, -2.597641, -0.773854, 1.570796, 1.702714],accel_mss,speed_ms,0,blend_radius_m)
    |   movel([0.131651, -1.340703, -2.597765, -0.773921, 1.570796, 1.702447],accel_mss,speed_ms,0,blend_radius_m)
    |   movel([0.132106, -1.340258, -2.598054, -0.774076, 1.570796, 1.702902],accel_mss,speed_ms,0,blend_radius_m)
    |   movel([0.132430, -1.340052, -2.598188, -0.774149, 1.570796, 1.703227],accel_mss,speed_ms,0,blend_radius_m)
    |   movel([0.132572, -1.339811, -2.598345, -0.774233, 1.570796, 1.703368],accel_mss,speed_ms,0,blend_radius_m)
    |   movel([0.132296, -1.339674, -2.598433, -0.774281, 1.570796, 1.703093],accel_mss,speed_ms,0,blend_radius_m)
    |   movel([0.132431, -1.339196, -2.598743, -0.774449, 1.570796, 1.703227],accel_mss,speed_ms,0,blend_radius_m)
    |   movel([0.132665, -1.338954, -2.598900, -0.774535, 1.570796, 1.703462],accel_mss,speed_ms,0,blend_radius_m)
    |   movel([0.133142, -1.338621, -2.599116, -0.774652, 1.570796, 1.703938],accel_mss,speed_ms,0,blend_radius_m)
    |   movel([0.133515, -1.338463, -2.599218, -0.774708, 1.570796, 1.704311],accel_mss,speed_ms,0,blend_radius_m)
    |   movel([0.133874, -1.338443, -2.599231, -0.774715, 1.570796, 1.704671],accel_mss,speed_ms,0,blend_radius_m)
    |   movel([0.134312, -1.338556, -2.599158, -0.774675, 1.570796, 1.705108],accel_mss,speed_ms,0,blend_radius_m)
    |   movel([0.134537, -1.338645, -2.599101, -0.774644, 1.570796, 1.705333],accel_mss,speed_ms,0,blend_radius_m)
    |   movel([0.134724, -1.338732, -2.599044, -0.774613, 1.570796, 1.705520],accel_mss,speed_ms,0,blend_radius_m)
    |   movel([0.134889, -1.338852, -2.598966, -0.774570, 1.570796, 1.705685],accel_mss,speed_ms,0,blend_radius_m)
    |   movel([0.135058, -1.339061, -2.598831, -0.774497, 1.570796, 1.705854],accel_mss,speed_ms,0,blend_radius_m)
    |   movel([0.135120, -1.339390, -2.598618, -0.774381, 1.570796, 1.705917],accel_mss,speed_ms,0,blend_radius_m)
    |   movel([0.134596, -1.339904, -2.598284, -0.774201, 1.570796, 1.705392],accel_mss,speed_ms,0,blend_radius_m)
    |   movel([0.134152, -1.340236, -2.598069, -0.774084, 1.570796, 1.704948],accel_mss,speed_ms,0,blend_radius_m)
    |   movel([0.134394, -1.340409, -2.597957, -0.774024, 1.570796, 1.705190],accel_mss,speed_ms,0,blend_radius_m)
    |   movel([0.134638, -1.340583, -2.597843, -0.773963, 1.570796, 1.705434],accel_mss,speed_ms,0,blend_radius_m)
    |   movel([0.134303, -1.340887, -2.597646, -0.773856, 1.570796, 1.705100],accel_mss,speed_ms,0,blend_radius_m)
    |   movel([0.133995, -1.341122, -2.597493, -0.773774, 1.570796, 1.704791],accel_mss,speed_ms,0,blend_radius_m)
    |   movel([0.133724, -1.341260, -2.597403, -0.773726, 1.570796, 1.704520],accel_mss,speed_ms,0,blend_radius_m)
    |   movel([0.133806, -1.341542, -2.597219, -0.773628, 1.570796, 1.704602],accel_mss,speed_ms,0,blend_radius_m)
    |   movel([0.134102, -1.341551, -2.597214, -0.773625, 1.570796, 1.704899],accel_mss,speed_ms,0,blend_radius_m)
    |   movel([0.134405, -1.341598, -2.597183, -0.773608, 1.570796, 1.705202],accel_mss,speed_ms,0,blend_radius_m)
    |   movel([0.134632, -1.341752, -2.597083, -0.773554, 1.570796, 1.705428],accel_mss,speed_ms,0,blend_radius_m)
    |   movel([0.134781, -1.341889, -2.596993, -0.773507, 1.570796, 1.705577],accel_mss,speed_ms,0,blend_radius_m)
    |   movel([0.134990, -1.341997, -2.596923, -0.773469, 1.570796, 1.705786],accel_mss,speed_ms,0,blend_radius_m)
    |   movel([0.134941, -1.342299, -2.596726, -0.773364, 1.570796, 1.705737],accel_mss,speed_ms,0,blend_radius_m)
    |   movel([0.134735, -1.342517, -2.596584, -0.773288, 1.570796, 1.705532],accel_mss,speed_ms,0,blend_radius_m)
    |   movel([0.134593, -1.342795, -2.596402, -0.773192, 1.570796, 1.705389],accel_mss,speed_ms,0,blend_radius_m)
    |   movel([0.134351, -1.343086, -2.596212, -0.773091, 1.570796, 1.705148],accel_mss,speed_ms,0,blend_radius_m)
    |   movel([0.134008, -1.343305, -2.596069, -0.773015, 1.570796, 1.704805],accel_mss,speed_ms,0,blend_radius_m)
    |   movel([0.133511, -1.343459, -2.595968, -0.772961, 1.570796, 1.704307],accel_mss,speed_ms,0,blend_radius_m)
    |   speed_ms = 0.003
    |   movel([0.133372, -1.346971, -2.597436, -0.767983, 1.570796, 1.704169],accel_mss,speed_ms,0,blend_radius_m)
    |   speed_ms = 0.007
    |   movel([0.133523, -1.347193, -2.597289, -0.767907, 1.570796, 1.704320],accel_mss,speed_ms,0,blend_radius_m)
    |   movel([0.133757, -1.347298, -2.597220, -0.767871, 1.570796, 1.704553],accel_mss,speed_ms,0,blend_radius_m)
    |   movel([0.133786, -1.347602, -2.597020, -0.767767, 1.570796, 1.704582],accel_mss,speed_ms,0,blend_radius_m)
    |   movel([0.133733, -1.347914, -2.596815, -0.767660, 1.570796, 1.704530],accel_mss,speed_ms,0,blend_radius_m)
    |   movel([0.133693, -1.348161, -2.596652, -0.767576, 1.570796, 1.704490],accel_mss,speed_ms,0,blend_radius_m)
    |   movel([0.133685, -1.348509, -2.596422, -0.767457, 1.570796, 1.704481],accel_mss,speed_ms,0,blend_radius_m)
    |   movel([0.133764, -1.348693, -2.596301, -0.767395, 1.570796, 1.704561],accel_mss,speed_ms,0,blend_radius_m)
    |   movel([0.133678, -1.349146, -2.596002, -0.767241, 1.570796, 1.704474],accel_mss,speed_ms,0,blend_radius_m)
    |   movel([0.133620, -1.349397, -2.595836, -0.767156, 1.570796, 1.704416],accel_mss,speed_ms,0,blend_radius_m)
    |   movel([0.133584, -1.349783, -2.595581, -0.767025, 1.570796, 1.704380],accel_mss,speed_ms,0,blend_radius_m)
    |   movel([0.133696, -1.349958, -2.595466, -0.766966, 1.570796, 1.704493],accel_mss,speed_ms,0,blend_radius_m)
    |   movel([0.133614, -1.350596, -2.595043, -0.766750, 1.570796, 1.704411],accel_mss,speed_ms,0,blend_radius_m)
    |   movel([0.133501, -1.351244, -2.594614, -0.766532, 1.570796, 1.704297],accel_mss,speed_ms,0,blend_radius_m)
    |   movel([0.133318, -1.351501, -2.594443, -0.766445, 1.570796, 1.704114],accel_mss,speed_ms,0,blend_radius_m)
    |   movel([0.133224, -1.351989, -2.594119, -0.766281, 1.570796, 1.704020],accel_mss,speed_ms,0,blend_radius_m)
    |   movel([0.133196, -1.352302, -2.593911, -0.766176, 1.570796, 1.703993],accel_mss,speed_ms,0,blend_radius_m)
    |   movel([0.133171, -1.352618, -2.593701, -0.766070, 1.570796, 1.703967],accel_mss,speed_ms,0,blend_radius_m)
    |   movel([0.133130, -1.352872, -2.593532, -0.765985, 1.570796, 1.703926],accel_mss,speed_ms,0,blend_radius_m)
    |   movel([0.133029, -1.353111, -2.593372, -0.765905, 1.570796, 1.703825],accel_mss,speed_ms,0,blend_radius_m)
    |   movel([0.132912, -1.353375, -2.593197, -0.765817, 1.570796, 1.703709],accel_mss,speed_ms,0,blend_radius_m)
    |   movel([0.132787, -1.354205, -2.592644, -0.765541, 1.570796, 1.703583],accel_mss,speed_ms,0,blend_radius_m)
    |   movel([0.132241, -1.355938, -2.591485, -0.764967, 1.570796, 1.703037],accel_mss,speed_ms,0,blend_radius_m)
    |   movel([0.131630, -1.357780, -2.590248, -0.764361, 1.570796, 1.702426],accel_mss,speed_ms,0,blend_radius_m)
